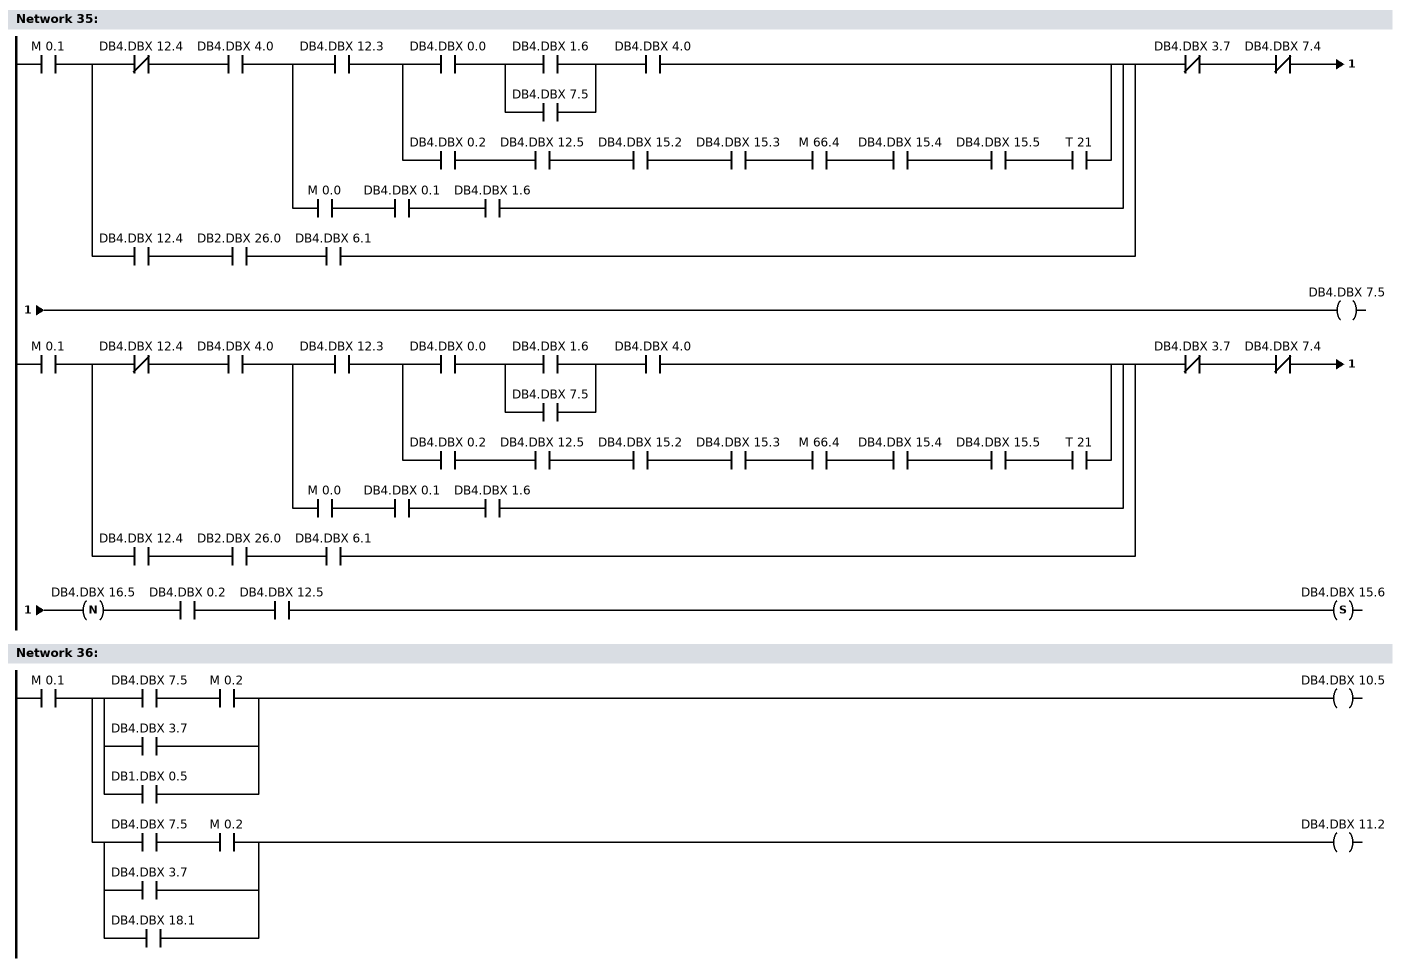
NETWORK
TITLE =
      A     M 0.1;
      A(;
      AN    DB4.DBX 12.4;
      A     DB4.DBX 4.0;
      A(;
      A     DB4.DBX 12.3;
      A(;
      A     DB4.DBX 0.0;
      A(;
      O     DB4.DBX 1.6;
      O     DB4.DBX 7.5;
      );
      A     DB4.DBX 4.0;
      O;
      A     DB4.DBX 0.2;
      A     DB4.DBX 12.5;
      A     DB4.DBX 15.2;
      A     DB4.DBX 15.3;
      A     M 66.4;
      A     DB4.DBX 15.4;
      A     DB4.DBX 15.5;
      A     T 21;
      );
      O;
      A     M 0.0;
      A     DB4.DBX 0.1;
      A     DB4.DBX 1.6;
      );
      O;
      A     DB4.DBX 12.4;
      A     DB2.DBX 26.0;
      A     DB4.DBX 6.1;
      );
      AN    DB4.DBX 3.7;
      AN    DB4.DBX 7.4;
      =     L 0.0;
      A     L 0.0;
      BLD   102;
      =     DB4.DBX 7.5;
      A(;
      A     L 0.0;
      FN    DB4.DBX 16.5;
      );
      A     DB4.DBX 0.2;
      A     DB4.DBX 12.5;
      S     DB4.DBX 15.6;
NETWORK
TITLE =
      A     M 0.1;
      =     L 0.0;
      A     L 0.0;
      A(;
      A     DB4.DBX 7.5;
      A     M 0.2;
      O     DB4.DBX 3.7;
      O     DB1.DBX 0.5;
      );
      =     DB4.DBX 10.5;
      A     L 0.0;
      A(;
      A     DB4.DBX 7.5;
      A     M 0.2;
      O     DB4.DBX 3.7;
      O     DB4.DBX 18.1;
      );
      =     DB4.DBX 11.2;
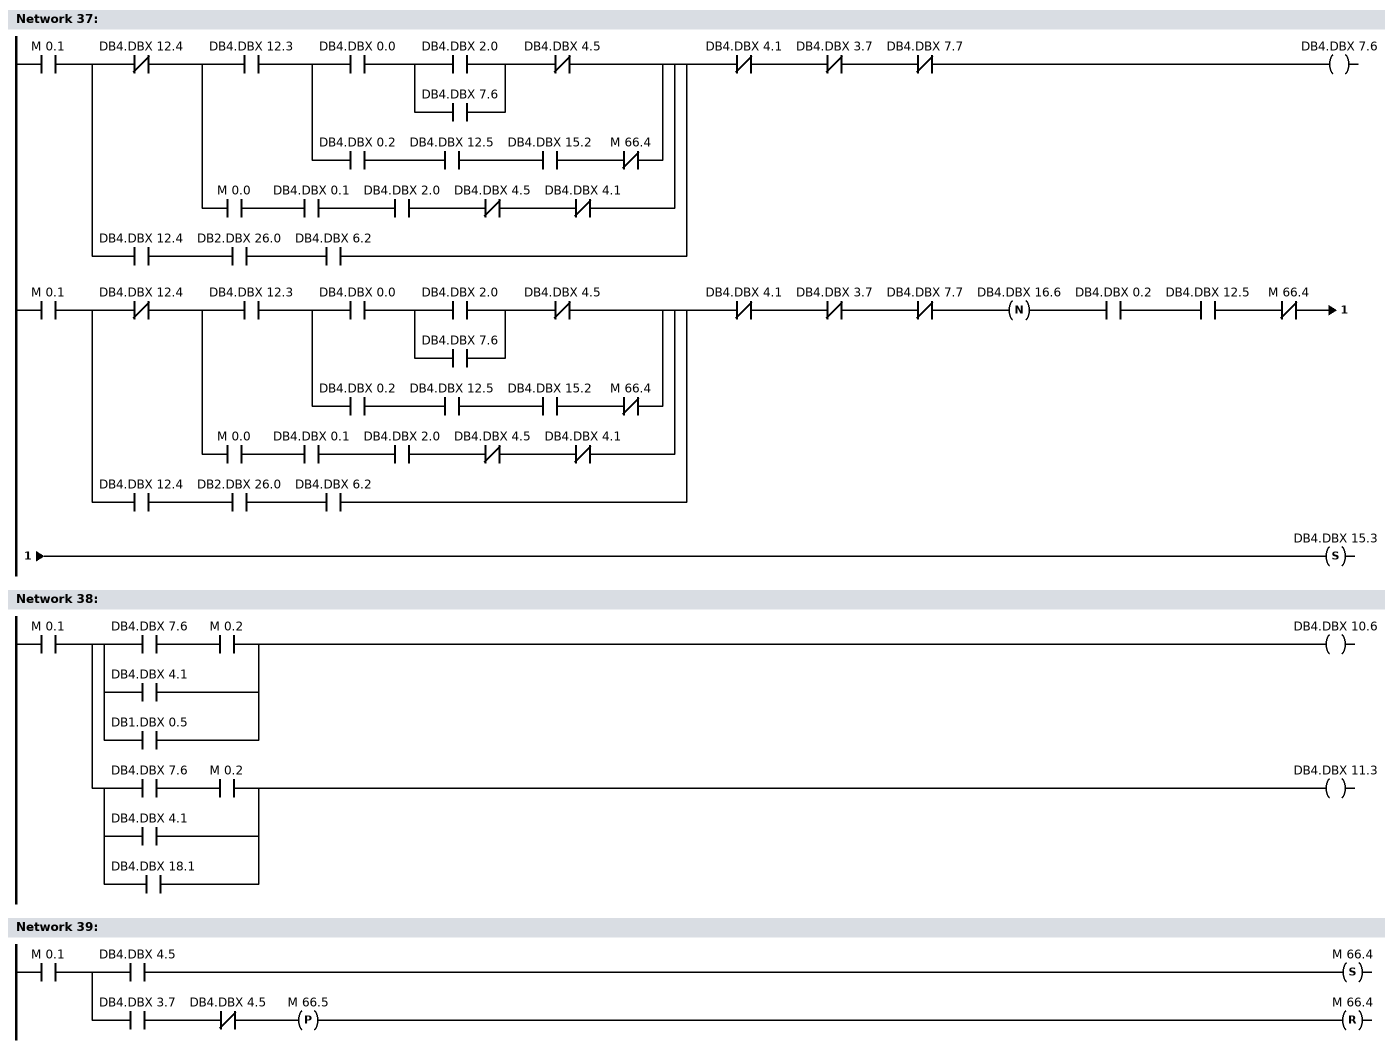
NETWORK
TITLE =
      A     M 0.1;
      A(;
      AN    DB4.DBX 12.4;
      A(;
      A     DB4.DBX 12.3;
      A(;
      A     DB4.DBX 0.0;
      A(;
      O     DB4.DBX 2.0;
      O     DB4.DBX 7.6;
      );
      AN    DB4.DBX 4.5;
      O;
      A     DB4.DBX 0.2;
      A     DB4.DBX 12.5;
      A     DB4.DBX 15.2;
      AN    M 66.4;
      );
      O;
      A     M 0.0;
      A     DB4.DBX 0.1;
      A     DB4.DBX 2.0;
      AN    DB4.DBX 4.5;
      AN    DB4.DBX 4.1;
      );
      O;
      A     DB4.DBX 12.4;
      A     DB2.DBX 26.0;
      A     DB4.DBX 6.2;
      );
      AN    DB4.DBX 4.1;
      AN    DB4.DBX 3.7;
      AN    DB4.DBX 7.7;
      =     L 0.0;
      A     L 0.0;
      BLD   102;
      =     DB4.DBX 7.6;
      A(;
      A     L 0.0;
      FN    DB4.DBX 16.6;
      );
      A     DB4.DBX 0.2;
      A     DB4.DBX 12.5;
      AN    M 66.4;
      S     DB4.DBX 15.3;
NETWORK
TITLE =
      A     M 0.1;
      =     L 0.0;
      A     L 0.0;
      A(;
      A     DB4.DBX 7.6;
      A     M 0.2;
      O     DB4.DBX 4.1;
      O     DB1.DBX 0.5;
      );
      =     DB4.DBX 10.6;
      A     L 0.0;
      A(;
      A     DB4.DBX 7.6;
      A     M 0.2;
      O     DB4.DBX 4.1;
      O     DB4.DBX 18.1;
      );
      =     DB4.DBX 11.3;
NETWORK
TITLE =
      A     M 0.1;
      =     L 0.0;
      A     L 0.0;
      A     DB4.DBX 4.5;
      S     M 66.4;
      A     L 0.0;
      A     DB4.DBX 3.7;
      AN    DB4.DBX 4.5;
      FP    M 66.5;
      R     M 66.4;
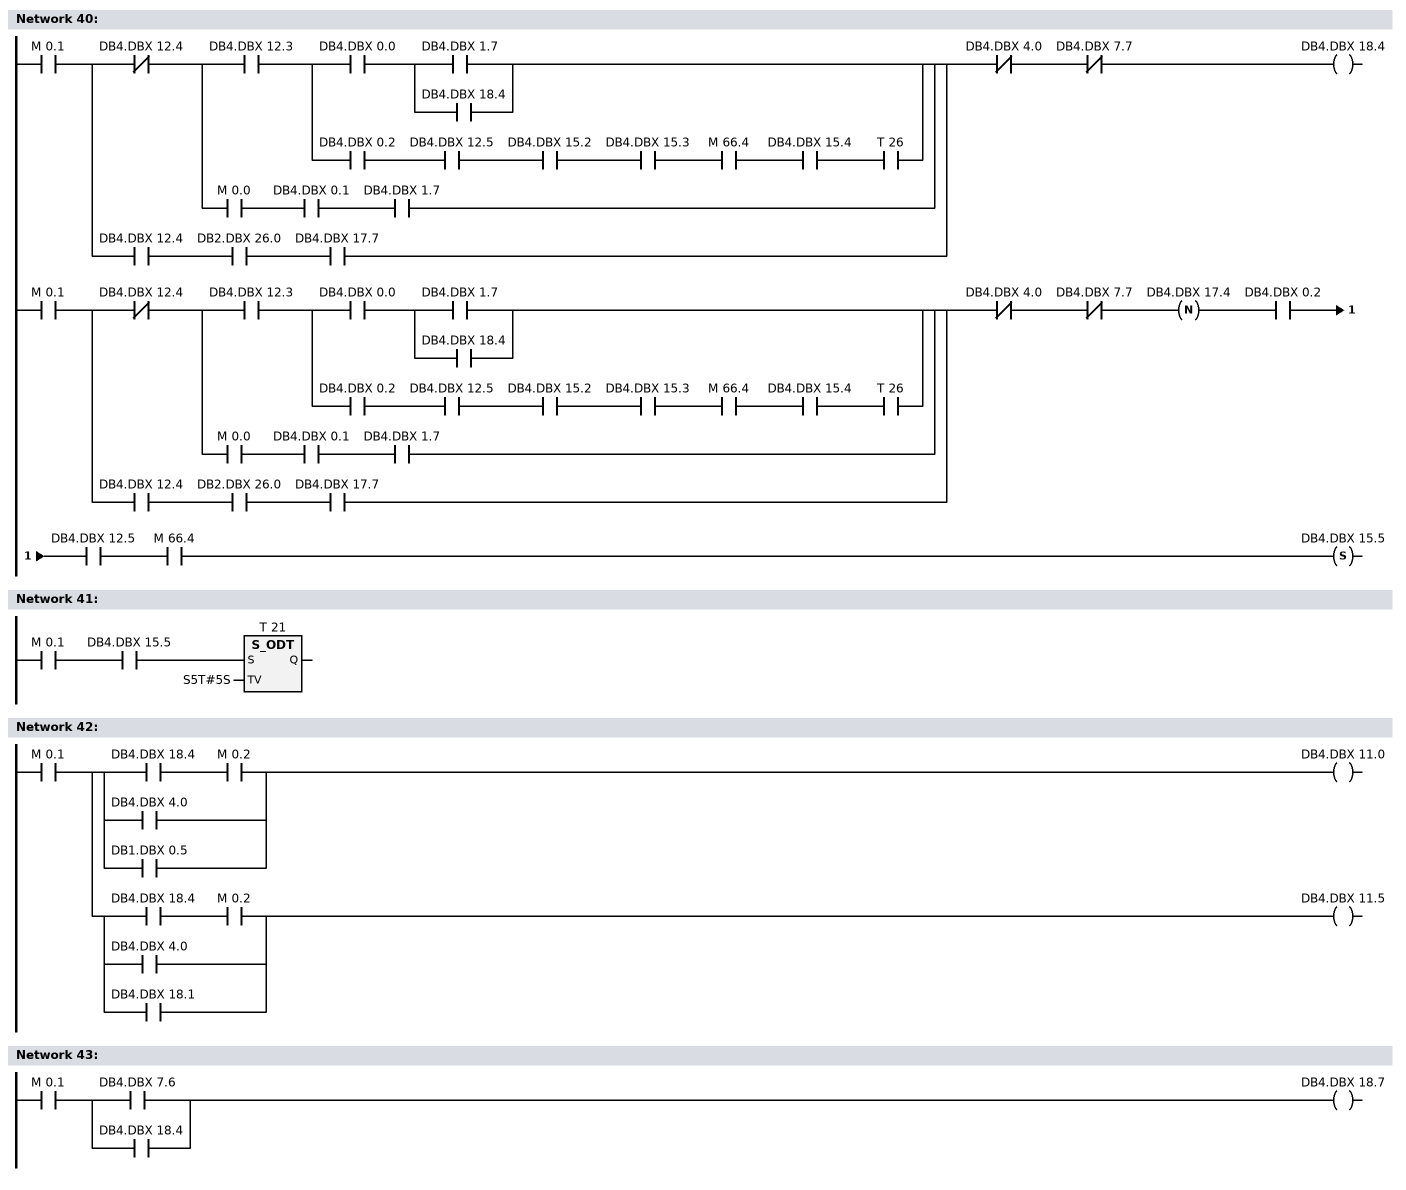
NETWORK
TITLE =
      A     M 0.1;
      A(;
      AN    DB4.DBX 12.4;
      A(;
      A     DB4.DBX 12.3;
      A(;
      A     DB4.DBX 0.0;
      A(;
      O     DB4.DBX 1.7;
      O     DB4.DBX 18.4;
      );
      O;
      A     DB4.DBX 0.2;
      A     DB4.DBX 12.5;
      A     DB4.DBX 15.2;
      A     DB4.DBX 15.3;
      A     M 66.4;
      A     DB4.DBX 15.4;
      A     T 26;
      );
      O;
      A     M 0.0;
      A     DB4.DBX 0.1;
      A     DB4.DBX 1.7;
      );
      O;
      A     DB4.DBX 12.4;
      A     DB2.DBX 26.0;
      A     DB4.DBX 17.7;
      );
      AN    DB4.DBX 4.0;
      AN    DB4.DBX 7.7;
      =     L 0.0;
      A     L 0.0;
      BLD   102;
      =     DB4.DBX 18.4;
      A(;
      A     L 0.0;
      FN    DB4.DBX 17.4;
      );
      A     DB4.DBX 0.2;
      A     DB4.DBX 12.5;
      A     M 66.4;
      S     DB4.DBX 15.5;
NETWORK
TITLE =
      A     M 0.1;
      A     DB4.DBX 15.5;
      L     S5T#5S;
      SD    T 21;
      NOP   0;
      NOP   0;
      NOP   0;
      NOP   0;
NETWORK
TITLE =
      A     M 0.1;
      =     L 0.0;
      A     L 0.0;
      A(;
      A     DB4.DBX 18.4;
      A     M 0.2;
      O     DB4.DBX 4.0;
      O     DB1.DBX 0.5;
      );
      =     DB4.DBX 11.0;
      A     L 0.0;
      A(;
      A     DB4.DBX 18.4;
      A     M 0.2;
      O     DB4.DBX 4.0;
      O     DB4.DBX 18.1;
      );
      =     DB4.DBX 11.5;
NETWORK
TITLE =
      A     M 0.1;
      A(;
      O     DB4.DBX 7.6;
      O     DB4.DBX 18.4;
      );
      =     DB4.DBX 18.7;
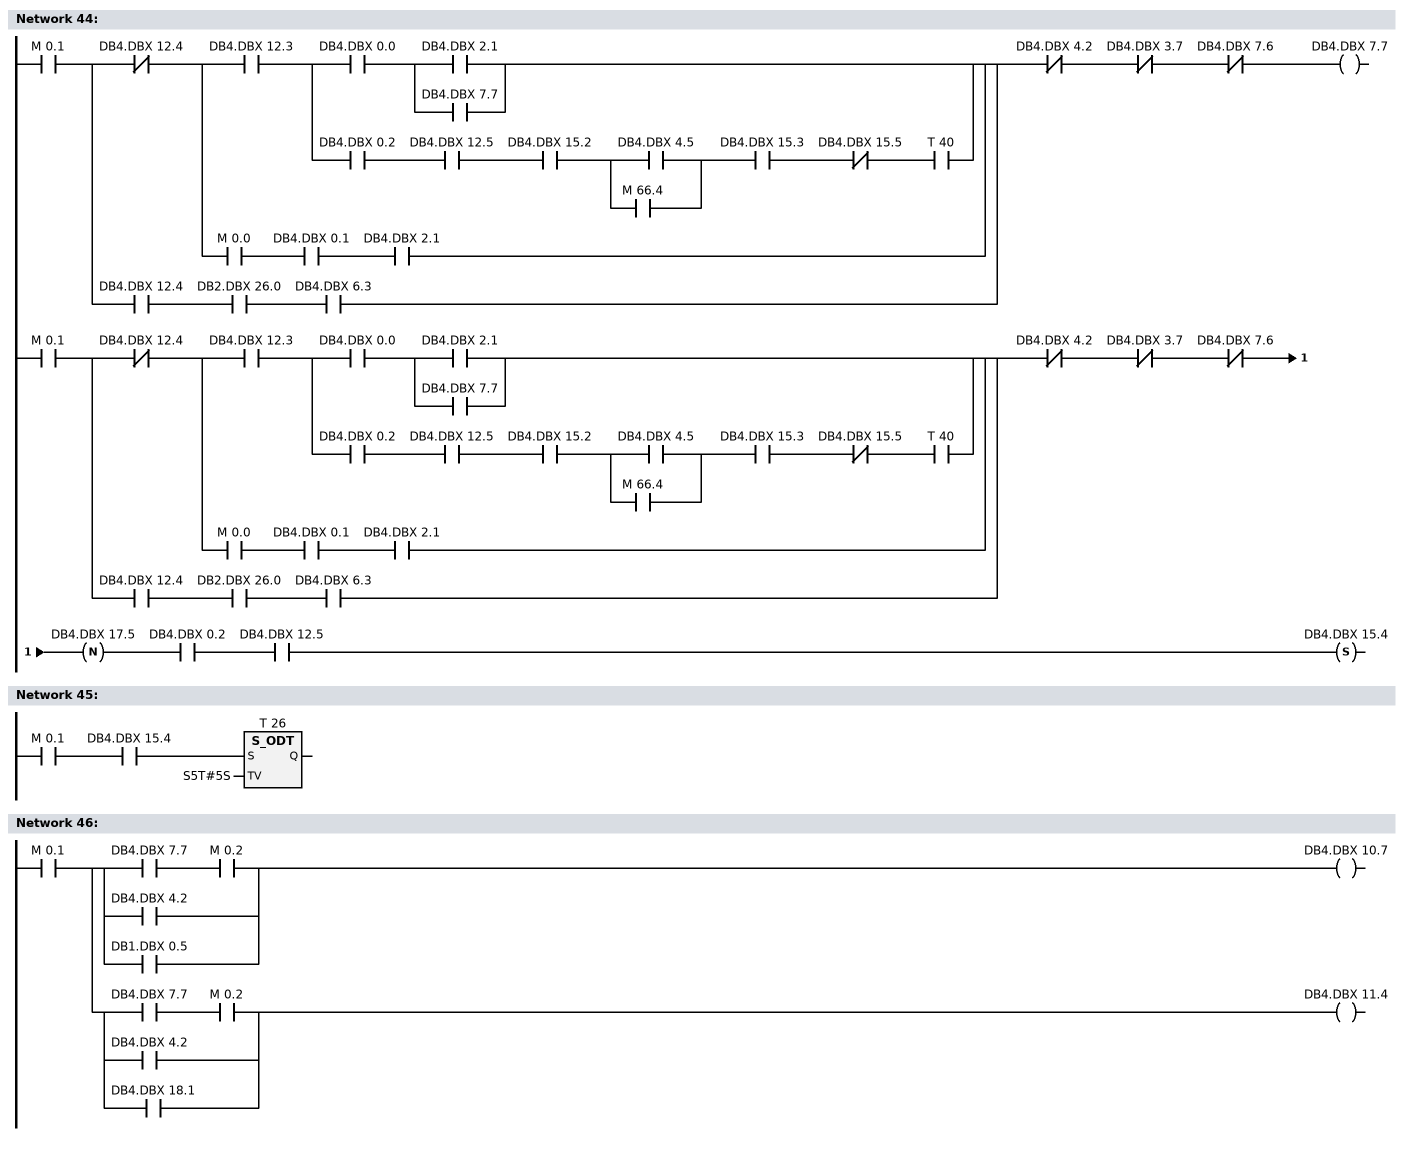
NETWORK
TITLE =
      A     M 0.1;
      A(;
      AN    DB4.DBX 12.4;
      A(;
      A     DB4.DBX 12.3;
      A(;
      A     DB4.DBX 0.0;
      A(;
      O     DB4.DBX 2.1;
      O     DB4.DBX 7.7;
      );
      O;
      A     DB4.DBX 0.2;
      A     DB4.DBX 12.5;
      A     DB4.DBX 15.2;
      A(;
      O     DB4.DBX 4.5;
      O     M 66.4;
      );
      A     DB4.DBX 15.3;
      AN    DB4.DBX 15.5;
      A     T 40;
      );
      O;
      A     M 0.0;
      A     DB4.DBX 0.1;
      A     DB4.DBX 2.1;
      );
      O;
      A     DB4.DBX 12.4;
      A     DB2.DBX 26.0;
      A     DB4.DBX 6.3;
      );
      AN    DB4.DBX 4.2;
      AN    DB4.DBX 3.7;
      AN    DB4.DBX 7.6;
      =     L 0.0;
      A     L 0.0;
      BLD   102;
      =     DB4.DBX 7.7;
      A(;
      A     L 0.0;
      FN    DB4.DBX 17.5;
      );
      A     DB4.DBX 0.2;
      A     DB4.DBX 12.5;
      S     DB4.DBX 15.4;
NETWORK
TITLE =
      A     M 0.1;
      A     DB4.DBX 15.4;
      L     S5T#5S;
      SD    T 26;
      NOP   0;
      NOP   0;
      NOP   0;
      NOP   0;
NETWORK
TITLE =
      A     M 0.1;
      =     L 0.0;
      A     L 0.0;
      A(;
      A     DB4.DBX 7.7;
      A     M 0.2;
      O     DB4.DBX 4.2;
      O     DB1.DBX 0.5;
      );
      =     DB4.DBX 10.7;
      A     L 0.0;
      A(;
      A     DB4.DBX 7.7;
      A     M 0.2;
      O     DB4.DBX 4.2;
      O     DB4.DBX 18.1;
      );
      =     DB4.DBX 11.4;
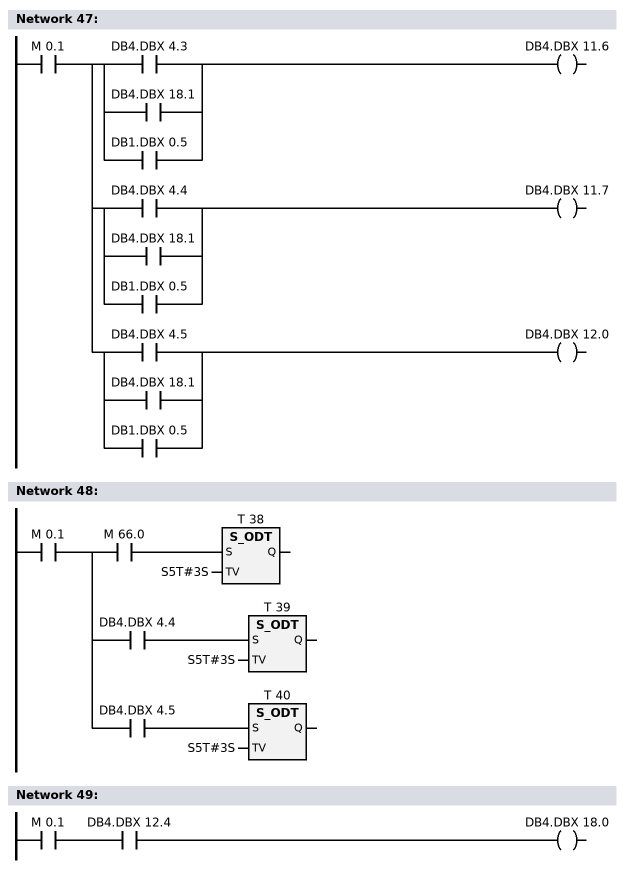
NETWORK
TITLE =
      A     M 0.1;
      =     L 0.0;
      A     L 0.0;
      A(;
      O     DB4.DBX 4.3;
      O     DB4.DBX 18.1;
      O     DB1.DBX 0.5;
      );
      =     DB4.DBX 11.6;
      A     L 0.0;
      A(;
      O     DB4.DBX 4.4;
      O     DB4.DBX 18.1;
      O     DB1.DBX 0.5;
      );
      =     DB4.DBX 11.7;
      A     L 0.0;
      A(;
      O     DB4.DBX 4.5;
      O     DB4.DBX 18.1;
      O     DB1.DBX 0.5;
      );
      =     DB4.DBX 12.0;
NETWORK
TITLE =
      A     M 0.1;
      =     L 0.0;
      A     L 0.0;
      A     M 66.0;
      L     S5T#3S;
      SD    T 38;
      NOP   0;
      NOP   0;
      NOP   0;
      NOP   0;
      A     L 0.0;
      A     DB4.DBX 4.4;
      L     S5T#3S;
      SD    T 39;
      NOP   0;
      NOP   0;
      NOP   0;
      NOP   0;
      A     L 0.0;
      A     DB4.DBX 4.5;
      L     S5T#3S;
      SD    T 40;
      NOP   0;
      NOP   0;
      NOP   0;
      NOP   0;
NETWORK
TITLE =
      A     M 0.1;
      A     DB4.DBX 12.4;
      =     DB4.DBX 18.0;
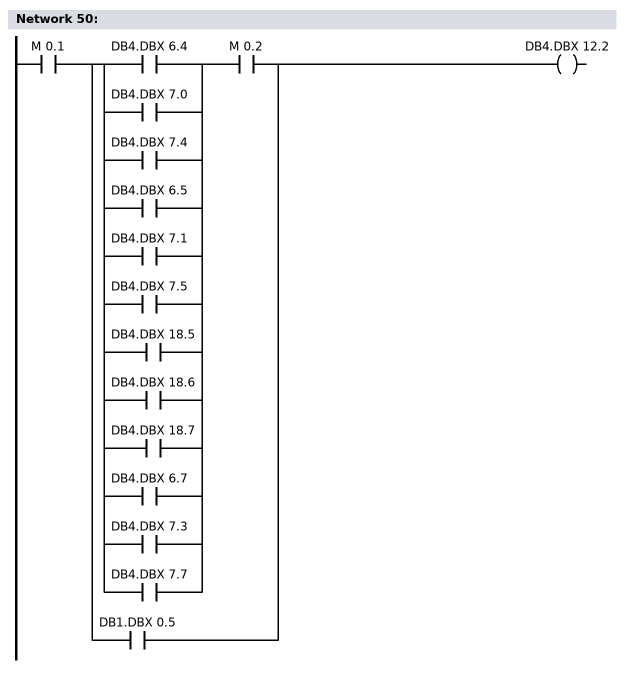
NETWORK
TITLE =
      A     M 0.1;
      A(;
      A(;
      O     DB4.DBX 6.4;
      O     DB4.DBX 7.0;
      O     DB4.DBX 7.4;
      O     DB4.DBX 6.5;
      O     DB4.DBX 7.1;
      O     DB4.DBX 7.5;
      O     DB4.DBX 18.5;
      O     DB4.DBX 18.6;
      O     DB4.DBX 18.7;
      O     DB4.DBX 6.7;
      O     DB4.DBX 7.3;
      O     DB4.DBX 7.7;
      );
      A     M 0.2;
      O     DB1.DBX 0.5;
      );
      =     DB4.DBX 12.2;
END_FUNCTION

FUNCTION FC 10 : VOID
AUTHOR : Arun_Ram
VERSION : 0.1
BEGIN
// (block stored without names or comments; labels and parameter names are numbered)
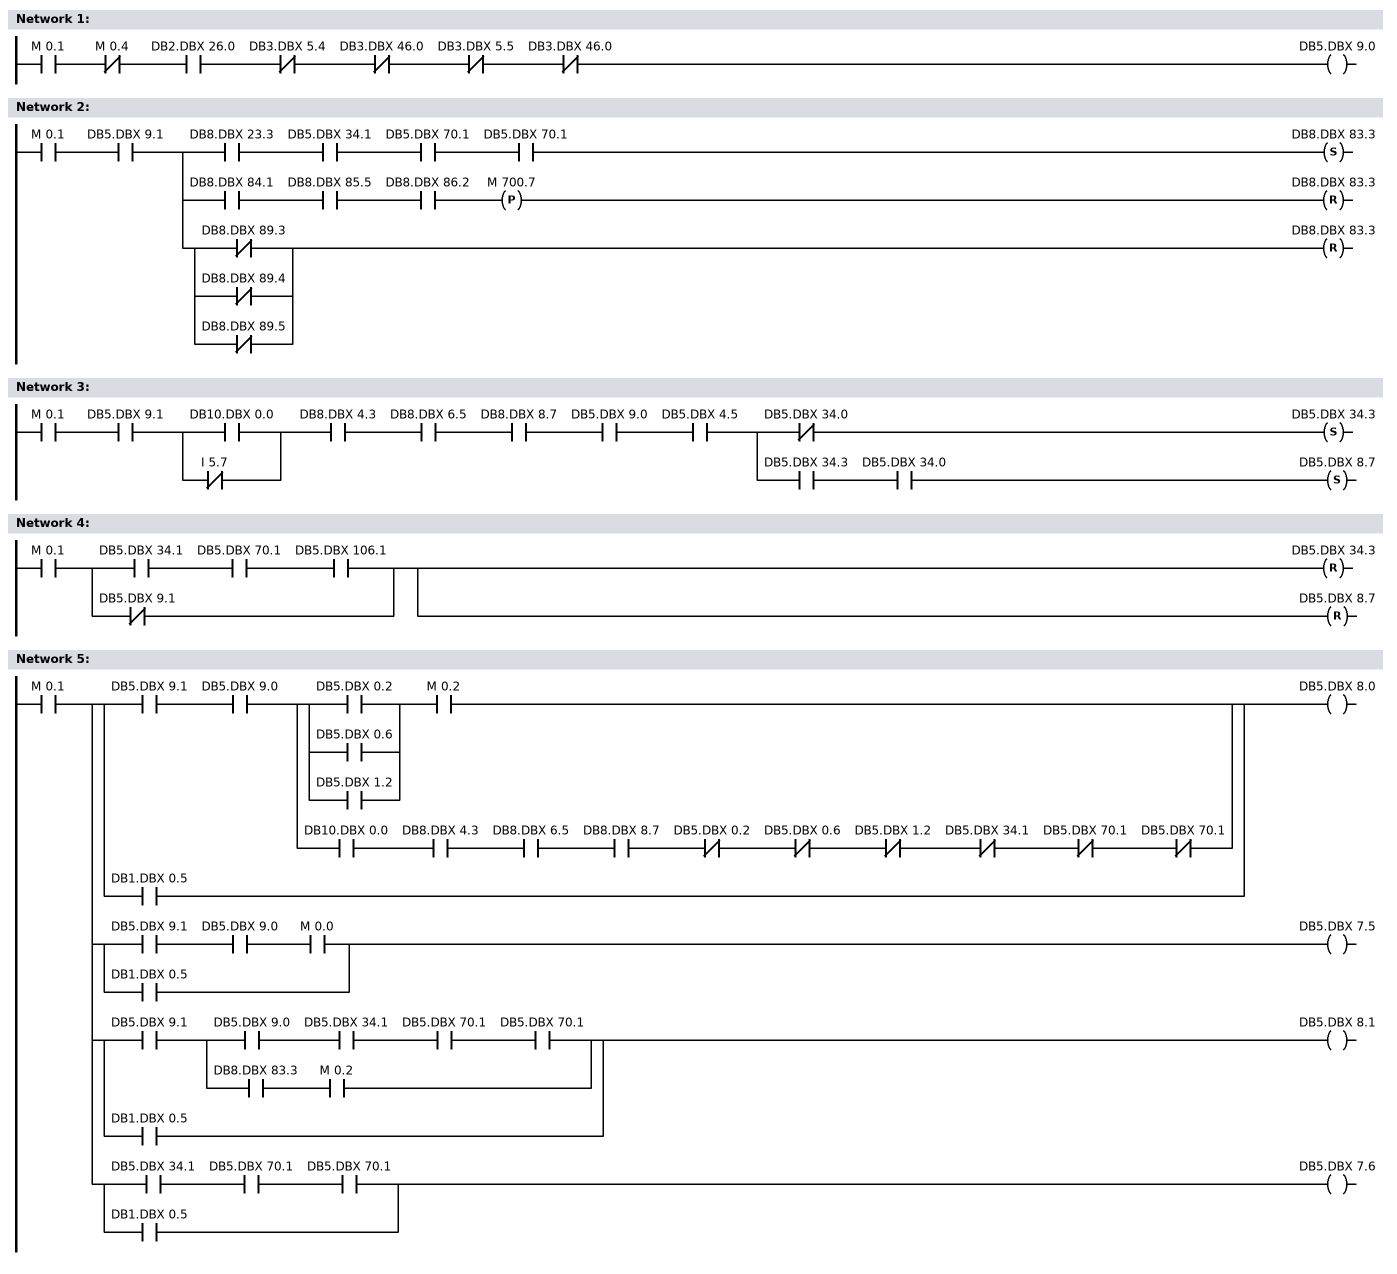
NETWORK
TITLE =
      A     M 0.1;
      AN    M 0.4;
      A     DB2.DBX 26.0;
      AN    DB3.DBX 5.4;
      AN    DB3.DBX 46.0;
      AN    DB3.DBX 5.5;
      AN    DB3.DBX 46.0;
      =     DB5.DBX 9.0;
NETWORK
TITLE =
      A     M 0.1;
      A     DB5.DBX 9.1;
      =     L 0.0;
      A     L 0.0;
      A     DB8.DBX 23.3;
      A     DB5.DBX 34.1;
      A     DB5.DBX 70.1;
      A     DB5.DBX 70.1;
      S     DB8.DBX 83.3;
      A     L 0.0;
      A     DB8.DBX 84.1;
      A     DB8.DBX 85.5;
      A     DB8.DBX 86.2;
      FP    M 700.7;
      R     DB8.DBX 83.3;
      A     L 0.0;
      A(;
      ON    DB8.DBX 89.3;
      ON    DB8.DBX 89.4;
      ON    DB8.DBX 89.5;
      );
      R     DB8.DBX 83.3;
NETWORK
TITLE =
      A     M 0.1;
      A     DB5.DBX 9.1;
      A(;
      O     DB10.DBX 0.0;
      ON    I 5.7;
      );
      A     DB8.DBX 4.3;
      A     DB8.DBX 6.5;
      A     DB8.DBX 8.7;
      A     DB5.DBX 9.0;
      A     DB5.DBX 4.5;
      =     L 0.0;
      A     L 0.0;
      AN    DB5.DBX 34.0;
      S     DB5.DBX 34.3;
      A     L 0.0;
      A     DB5.DBX 34.3;
      A     DB5.DBX 34.0;
      S     DB5.DBX 8.7;
NETWORK
TITLE =
      A     M 0.1;
      A(;
      A     DB5.DBX 34.1;
      A     DB5.DBX 70.1;
      A     DB5.DBX 106.1;
      ON    DB5.DBX 9.1;
      );
      R     DB5.DBX 34.3;
      R     DB5.DBX 8.7;
NETWORK
TITLE =
      A     M 0.1;
      =     L 0.0;
      A     L 0.0;
      A(;
      A     DB5.DBX 9.1;
      A     DB5.DBX 9.0;
      A(;
      A(;
      O     DB5.DBX 0.2;
      O     DB5.DBX 0.6;
      O     DB5.DBX 1.2;
      );
      A     M 0.2;
      O;
      A     DB10.DBX 0.0;
      A     DB8.DBX 4.3;
      A     DB8.DBX 6.5;
      A     DB8.DBX 8.7;
      AN    DB5.DBX 0.2;
      AN    DB5.DBX 0.6;
      AN    DB5.DBX 1.2;
      AN    DB5.DBX 34.1;
      AN    DB5.DBX 70.1;
      AN    DB5.DBX 70.1;
      );
      O     DB1.DBX 0.5;
      );
      =     DB5.DBX 8.0;
      A     L 0.0;
      A(;
      A     DB5.DBX 9.1;
      A     DB5.DBX 9.0;
      A     M 0.0;
      O     DB1.DBX 0.5;
      );
      =     DB5.DBX 7.5;
      A     L 0.0;
      A(;
      A     DB5.DBX 9.1;
      A(;
      A     DB5.DBX 9.0;
      A     DB5.DBX 34.1;
      A     DB5.DBX 70.1;
      A     DB5.DBX 70.1;
      O;
      A     DB8.DBX 83.3;
      A     M 0.2;
      );
      O     DB1.DBX 0.5;
      );
      =     DB5.DBX 8.1;
      A     L 0.0;
      A(;
      A     DB5.DBX 34.1;
      A     DB5.DBX 70.1;
      A     DB5.DBX 70.1;
      O     DB1.DBX 0.5;
      );
      =     DB5.DBX 7.6;
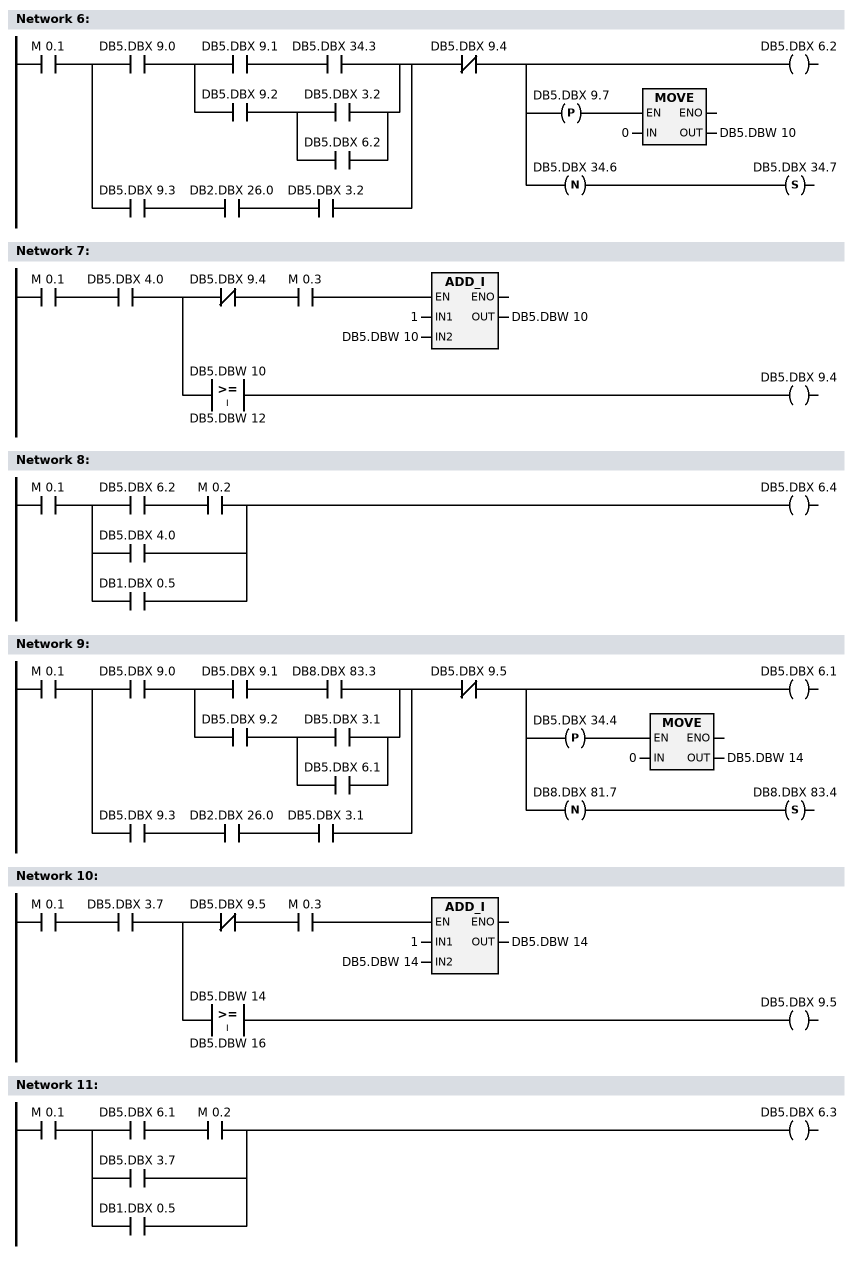
NETWORK
TITLE =
      A     M 0.1;
      A(;
      A     DB5.DBX 9.0;
      A(;
      A     DB5.DBX 9.1;
      A     DB5.DBX 34.3;
      O;
      A     DB5.DBX 9.2;
      A(;
      O     DB5.DBX 3.2;
      O     DB5.DBX 6.2;
      );
      );
      O;
      A     DB5.DBX 9.3;
      A     DB2.DBX 26.0;
      A     DB5.DBX 3.2;
      );
      AN    DB5.DBX 9.4;
      =     L 0.0;
      A     L 0.0;
      BLD   102;
      =     DB5.DBX 6.2;
      A     L 0.0;
      FP    DB5.DBX 9.7;
      JNB   M001;
      L     0;
      T     DB5.DBW 10;
M001: NOP   0;
      A     L 0.0;
      FN    DB5.DBX 34.6;
      S     DB5.DBX 34.7;
NETWORK
TITLE =
      A     M 0.1;
      A     DB5.DBX 4.0;
      =     L 0.0;
      A     L 0.0;
      AN    DB5.DBX 9.4;
      A     M 0.3;
      JNB   M002;
      L     1;
      L     DB5.DBW 10;
      +I;
      T     DB5.DBW 10;
M002: NOP   0;
      A     L 0.0;
      A(;
      L     DB5.DBW 10;
      L     DB5.DBW 12;
      >=I;
      );
      =     DB5.DBX 9.4;
NETWORK
TITLE =
      A     M 0.1;
      A(;
      A     DB5.DBX 6.2;
      A     M 0.2;
      O     DB5.DBX 4.0;
      O     DB1.DBX 0.5;
      );
      =     DB5.DBX 6.4;
NETWORK
TITLE =
      A     M 0.1;
      A(;
      A     DB5.DBX 9.0;
      A(;
      A     DB5.DBX 9.1;
      A     DB8.DBX 83.3;
      O;
      A     DB5.DBX 9.2;
      A(;
      O     DB5.DBX 3.1;
      O     DB5.DBX 6.1;
      );
      );
      O;
      A     DB5.DBX 9.3;
      A     DB2.DBX 26.0;
      A     DB5.DBX 3.1;
      );
      AN    DB5.DBX 9.5;
      =     L 0.0;
      A     L 0.0;
      BLD   102;
      =     DB5.DBX 6.1;
      A     L 0.0;
      FP    DB5.DBX 34.4;
      JNB   M003;
      L     0;
      T     DB5.DBW 14;
M003: NOP   0;
      A     L 0.0;
      FN    DB8.DBX 81.7;
      S     DB8.DBX 83.4;
NETWORK
TITLE =
      A     M 0.1;
      A     DB5.DBX 3.7;
      =     L 0.0;
      A     L 0.0;
      AN    DB5.DBX 9.5;
      A     M 0.3;
      JNB   M004;
      L     1;
      L     DB5.DBW 14;
      +I;
      T     DB5.DBW 14;
M004: NOP   0;
      A     L 0.0;
      A(;
      L     DB5.DBW 14;
      L     DB5.DBW 16;
      >=I;
      );
      =     DB5.DBX 9.5;
NETWORK
TITLE =
      A     M 0.1;
      A(;
      A     DB5.DBX 6.1;
      A     M 0.2;
      O     DB5.DBX 3.7;
      O     DB1.DBX 0.5;
      );
      =     DB5.DBX 6.3;
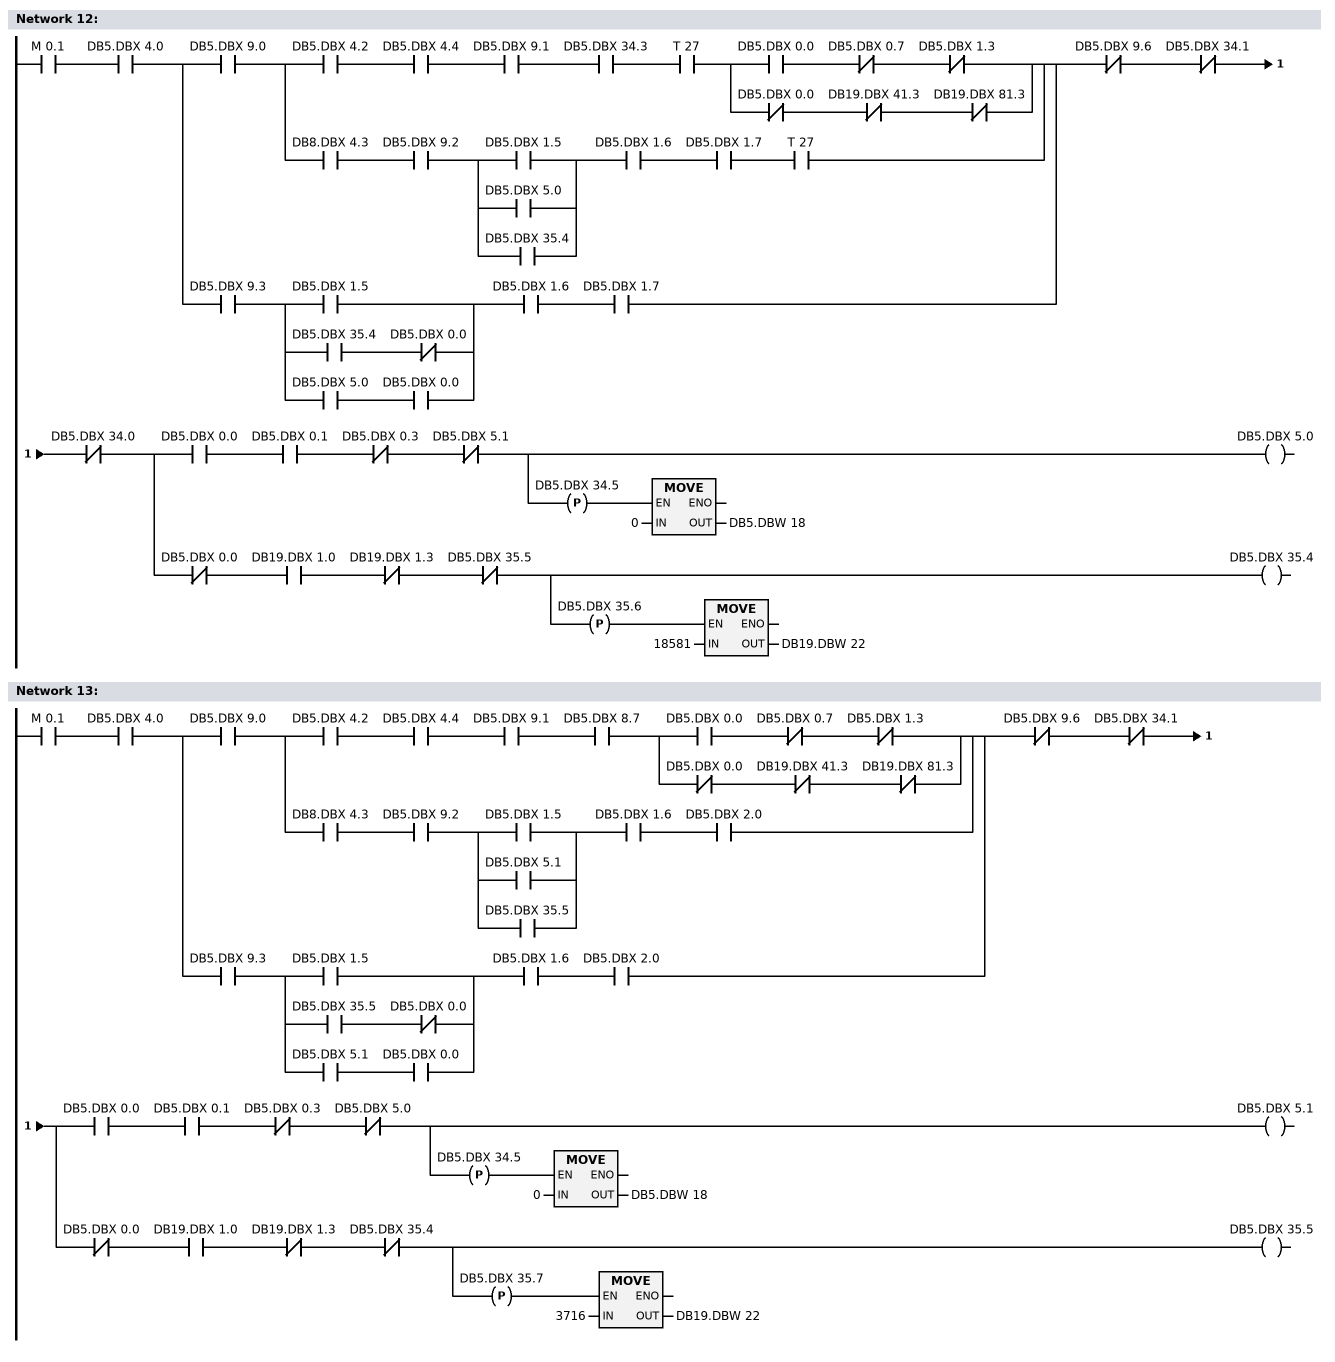
NETWORK
TITLE =
      A     M 0.1;
      A     DB5.DBX 4.0;
      A(;
      A     DB5.DBX 9.0;
      A(;
      A     DB5.DBX 4.2;
      A     DB5.DBX 4.4;
      A     DB5.DBX 9.1;
      A     DB5.DBX 34.3;
      A     T 27;
      A(;
      A     DB5.DBX 0.0;
      AN    DB5.DBX 0.7;
      AN    DB5.DBX 1.3;
      O;
      AN    DB5.DBX 0.0;
      AN    DB19.DBX 41.3;
      AN    DB19.DBX 81.3;
      );
      O;
      A     DB8.DBX 4.3;
      A     DB5.DBX 9.2;
      A(;
      O     DB5.DBX 1.5;
      O     DB5.DBX 5.0;
      O     DB5.DBX 35.4;
      );
      A     DB5.DBX 1.6;
      A     DB5.DBX 1.7;
      A     T 27;
      );
      O;
      A     DB5.DBX 9.3;
      A(;
      O     DB5.DBX 1.5;
      O;
      A     DB5.DBX 35.4;
      AN    DB5.DBX 0.0;
      O;
      A     DB5.DBX 5.0;
      A     DB5.DBX 0.0;
      );
      A     DB5.DBX 1.6;
      A     DB5.DBX 1.7;
      );
      AN    DB5.DBX 9.6;
      AN    DB5.DBX 34.1;
      AN    DB5.DBX 34.0;
      =     L 0.0;
      A     L 0.0;
      A     DB5.DBX 0.0;
      A     DB5.DBX 0.1;
      AN    DB5.DBX 0.3;
      AN    DB5.DBX 5.1;
      =     L 0.1;
      A     L 0.1;
      BLD   102;
      =     DB5.DBX 5.0;
      A     L 0.1;
      FP    DB5.DBX 34.5;
      JNB   M005;
      L     0;
      T     DB5.DBW 18;
M005: NOP   0;
      A     L 0.0;
      AN    DB5.DBX 0.0;
      A     DB19.DBX 1.0;
      AN    DB19.DBX 1.3;
      AN    DB5.DBX 35.5;
      =     L 0.1;
      A     L 0.1;
      BLD   102;
      =     DB5.DBX 35.4;
      A     L 0.1;
      FP    DB5.DBX 35.6;
      JNB   M006;
      L     18581;
      T     DB19.DBW 22;
M006: NOP   0;
NETWORK
TITLE =
      A     M 0.1;
      A     DB5.DBX 4.0;
      A(;
      A     DB5.DBX 9.0;
      A(;
      A     DB5.DBX 4.2;
      A     DB5.DBX 4.4;
      A     DB5.DBX 9.1;
      A     DB5.DBX 8.7;
      A(;
      A     DB5.DBX 0.0;
      AN    DB5.DBX 0.7;
      AN    DB5.DBX 1.3;
      O;
      AN    DB5.DBX 0.0;
      AN    DB19.DBX 41.3;
      AN    DB19.DBX 81.3;
      );
      O;
      A     DB8.DBX 4.3;
      A     DB5.DBX 9.2;
      A(;
      O     DB5.DBX 1.5;
      O     DB5.DBX 5.1;
      O     DB5.DBX 35.5;
      );
      A     DB5.DBX 1.6;
      A     DB5.DBX 2.0;
      );
      O;
      A     DB5.DBX 9.3;
      A(;
      O     DB5.DBX 1.5;
      O;
      A     DB5.DBX 35.5;
      AN    DB5.DBX 0.0;
      O;
      A     DB5.DBX 5.1;
      A     DB5.DBX 0.0;
      );
      A     DB5.DBX 1.6;
      A     DB5.DBX 2.0;
      );
      AN    DB5.DBX 9.6;
      AN    DB5.DBX 34.1;
      =     L 0.0;
      A     L 0.0;
      A     DB5.DBX 0.0;
      A     DB5.DBX 0.1;
      AN    DB5.DBX 0.3;
      AN    DB5.DBX 5.0;
      =     L 0.1;
      A     L 0.1;
      BLD   102;
      =     DB5.DBX 5.1;
      A     L 0.1;
      FP    DB5.DBX 34.5;
      JNB   M007;
      L     0;
      T     DB5.DBW 18;
M007: NOP   0;
      A     L 0.0;
      AN    DB5.DBX 0.0;
      A     DB19.DBX 1.0;
      AN    DB19.DBX 1.3;
      AN    DB5.DBX 35.4;
      =     L 0.1;
      A     L 0.1;
      BLD   102;
      =     DB5.DBX 35.5;
      A     L 0.1;
      FP    DB5.DBX 35.7;
      JNB   M008;
      L     3716;
      T     DB19.DBW 22;
M008: NOP   0;
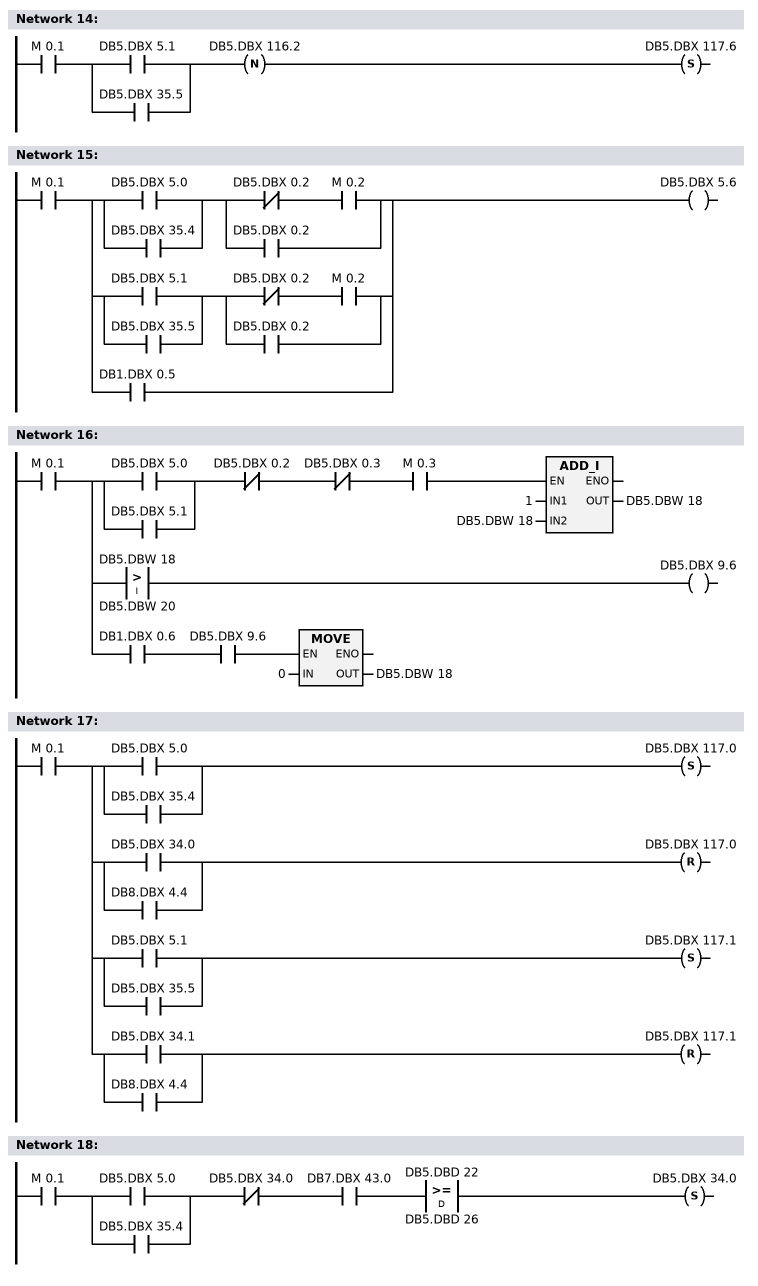
NETWORK
TITLE =
      A     M 0.1;
      A(;
      O     DB5.DBX 5.1;
      O     DB5.DBX 35.5;
      );
      FN    DB5.DBX 116.2;
      S     DB5.DBX 117.6;
NETWORK
TITLE =
      A     M 0.1;
      A(;
      A(;
      O     DB5.DBX 5.0;
      O     DB5.DBX 35.4;
      );
      A(;
      AN    DB5.DBX 0.2;
      A     M 0.2;
      O     DB5.DBX 0.2;
      );
      O;
      A(;
      O     DB5.DBX 5.1;
      O     DB5.DBX 35.5;
      );
      A(;
      AN    DB5.DBX 0.2;
      A     M 0.2;
      O     DB5.DBX 0.2;
      );
      O     DB1.DBX 0.5;
      );
      =     DB5.DBX 5.6;
NETWORK
TITLE =
      A     M 0.1;
      =     L 0.0;
      A     L 0.0;
      A(;
      O     DB5.DBX 5.0;
      O     DB5.DBX 5.1;
      );
      AN    DB5.DBX 0.2;
      AN    DB5.DBX 0.3;
      A     M 0.3;
      JNB   M009;
      L     1;
      L     DB5.DBW 18;
      +I;
      T     DB5.DBW 18;
M009: NOP   0;
      A     L 0.0;
      A(;
      L     DB5.DBW 18;
      L     DB5.DBW 20;
      >I;
      );
      =     DB5.DBX 9.6;
      A     L 0.0;
      A     DB1.DBX 0.6;
      A     DB5.DBX 9.6;
      JNB   M010;
      L     0;
      T     DB5.DBW 18;
M010: NOP   0;
NETWORK
TITLE =
      A     M 0.1;
      =     L 0.0;
      A     L 0.0;
      A(;
      O     DB5.DBX 5.0;
      O     DB5.DBX 35.4;
      );
      S     DB5.DBX 117.0;
      A     L 0.0;
      A(;
      O     DB5.DBX 34.0;
      O     DB8.DBX 4.4;
      );
      R     DB5.DBX 117.0;
      A     L 0.0;
      A(;
      O     DB5.DBX 5.1;
      O     DB5.DBX 35.5;
      );
      S     DB5.DBX 117.1;
      A     L 0.0;
      A(;
      O     DB5.DBX 34.1;
      O     DB8.DBX 4.4;
      );
      R     DB5.DBX 117.1;
NETWORK
TITLE =
      A     M 0.1;
      A(;
      O     DB5.DBX 5.0;
      O     DB5.DBX 35.4;
      );
      AN    DB5.DBX 34.0;
      A     DB7.DBX 43.0;
      A(;
      L     DB5.DBD 22;
      L     DB5.DBD 26;
      >=D;
      );
      S     DB5.DBX 34.0;
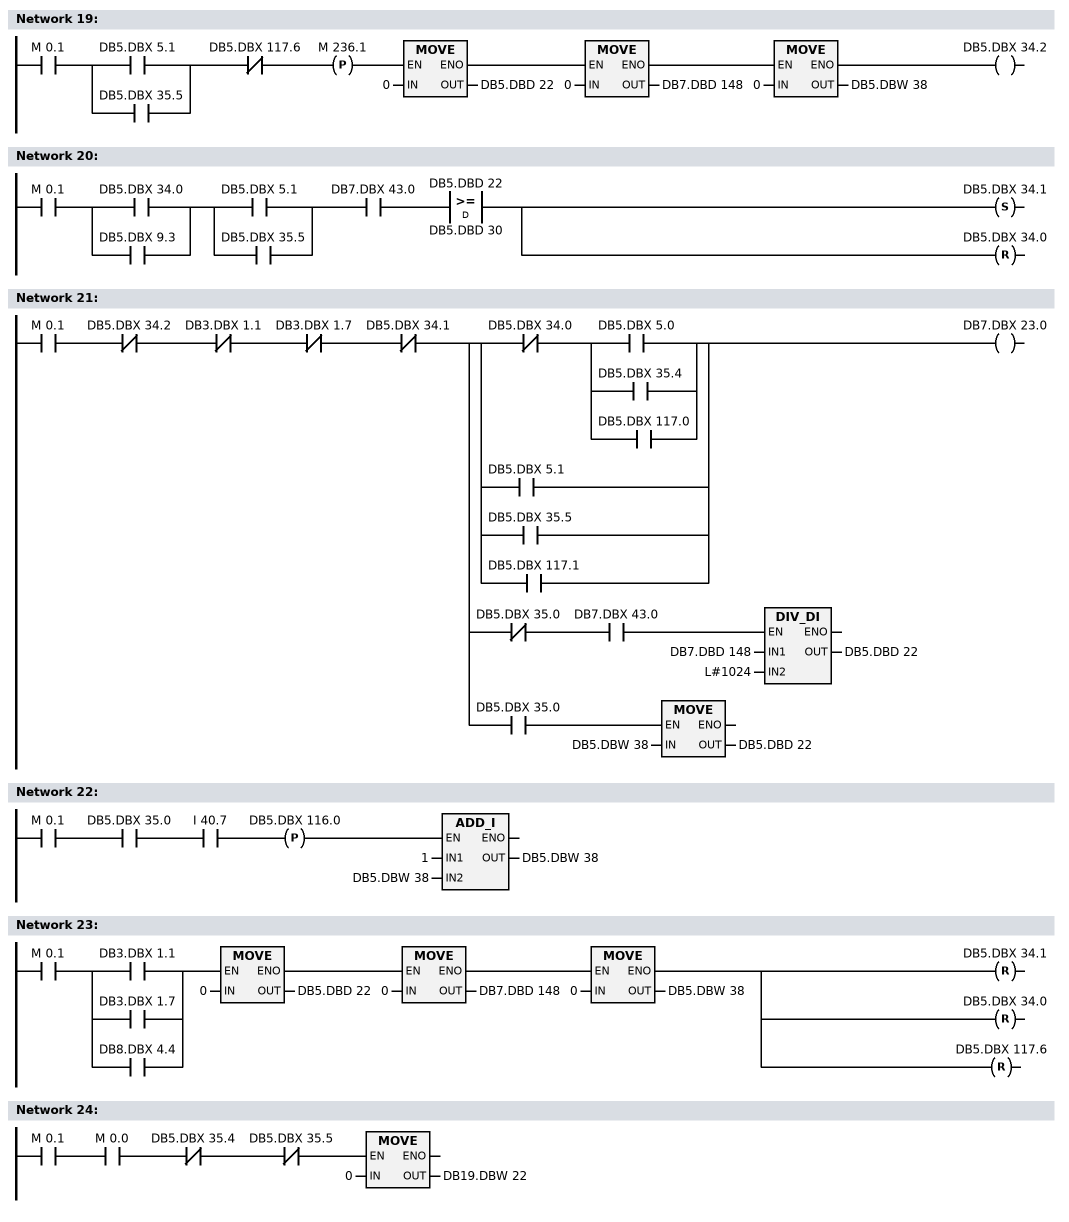
NETWORK
TITLE =
      A(;
      A(;
      A     M 0.1;
      A(;
      O     DB5.DBX 5.1;
      O     DB5.DBX 35.5;
      );
      AN    DB5.DBX 117.6;
      FP    M 236.1;
      JNB   M011;
      L     0;
      T     DB5.DBD 22;
      SET;
      SAVE;
      CLR;
M011: A     BR;
      );
      JNB   M012;
      L     0;
      T     DB7.DBD 148;
      SET;
      SAVE;
      CLR;
M012: A     BR;
      );
      JNB   M013;
      L     0;
      T     DB5.DBW 38;
      SET;
      SAVE;
      CLR;
M013: A     BR;
      =     DB5.DBX 34.2;
NETWORK
TITLE =
      A     M 0.1;
      A(;
      O     DB5.DBX 34.0;
      O     DB5.DBX 9.3;
      );
      A(;
      O     DB5.DBX 5.1;
      O     DB5.DBX 35.5;
      );
      A     DB7.DBX 43.0;
      A(;
      L     DB5.DBD 22;
      L     DB5.DBD 30;
      >=D;
      );
      S     DB5.DBX 34.1;
      R     DB5.DBX 34.0;
NETWORK
TITLE =
      A     M 0.1;
      AN    DB5.DBX 34.2;
      AN    DB3.DBX 1.1;
      AN    DB3.DBX 1.7;
      AN    DB5.DBX 34.1;
      =     L 0.0;
      A     L 0.0;
      A(;
      AN    DB5.DBX 34.0;
      A(;
      O     DB5.DBX 5.0;
      O     DB5.DBX 35.4;
      O     DB5.DBX 117.0;
      );
      O     DB5.DBX 5.1;
      O     DB5.DBX 35.5;
      O     DB5.DBX 117.1;
      );
      =     DB7.DBX 23.0;
      A     L 0.0;
      AN    DB5.DBX 35.0;
      A     DB7.DBX 43.0;
      JNB   M014;
      L     DB7.DBD 148;
      L     L#1024;
      /D;
      T     DB5.DBD 22;
M014: NOP   0;
      A     L 0.0;
      A     DB5.DBX 35.0;
      JNB   M015;
      L     DB5.DBW 38;
      T     DB5.DBD 22;
M015: NOP   0;
NETWORK
TITLE =
      A     M 0.1;
      A     DB5.DBX 35.0;
      A     I 40.7;
      FP    DB5.DBX 116.0;
      JNB   M016;
      L     1;
      L     DB5.DBW 38;
      +I;
      T     DB5.DBW 38;
M016: NOP   0;
NETWORK
TITLE =
      A(;
      A(;
      A     M 0.1;
      A(;
      O     DB3.DBX 1.1;
      O     DB3.DBX 1.7;
      O     DB8.DBX 4.4;
      );
      JNB   M017;
      L     0;
      T     DB5.DBD 22;
      SET;
      SAVE;
      CLR;
M017: A     BR;
      );
      JNB   M018;
      L     0;
      T     DB7.DBD 148;
      SET;
      SAVE;
      CLR;
M018: A     BR;
      );
      JNB   M019;
      L     0;
      T     DB5.DBW 38;
      SET;
      SAVE;
      CLR;
M019: A     BR;
      R     DB5.DBX 34.1;
      R     DB5.DBX 34.0;
      R     DB5.DBX 117.6;
NETWORK
TITLE =
      A     M 0.1;
      A     M 0.0;
      AN    DB5.DBX 35.4;
      AN    DB5.DBX 35.5;
      JNB   M020;
      L     0;
      T     DB19.DBW 22;
M020: NOP   0;
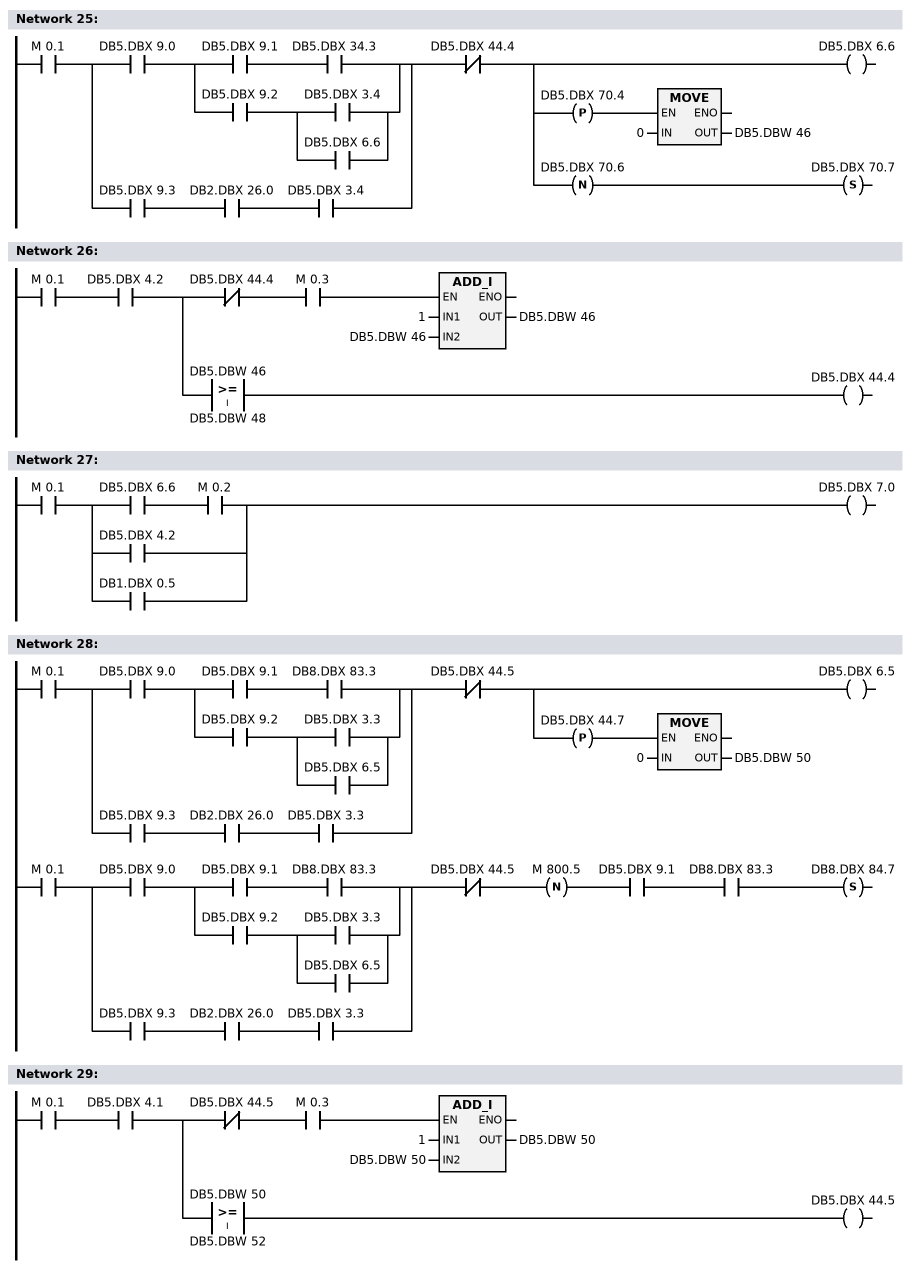
NETWORK
TITLE =
      A     M 0.1;
      A(;
      A     DB5.DBX 9.0;
      A(;
      A     DB5.DBX 9.1;
      A     DB5.DBX 34.3;
      O;
      A     DB5.DBX 9.2;
      A(;
      O     DB5.DBX 3.4;
      O     DB5.DBX 6.6;
      );
      );
      O;
      A     DB5.DBX 9.3;
      A     DB2.DBX 26.0;
      A     DB5.DBX 3.4;
      );
      AN    DB5.DBX 44.4;
      =     L 0.0;
      A     L 0.0;
      BLD   102;
      =     DB5.DBX 6.6;
      A     L 0.0;
      FP    DB5.DBX 70.4;
      JNB   M021;
      L     0;
      T     DB5.DBW 46;
M021: NOP   0;
      A     L 0.0;
      FN    DB5.DBX 70.6;
      S     DB5.DBX 70.7;
NETWORK
TITLE =
      A     M 0.1;
      A     DB5.DBX 4.2;
      =     L 0.0;
      A     L 0.0;
      AN    DB5.DBX 44.4;
      A     M 0.3;
      JNB   M022;
      L     1;
      L     DB5.DBW 46;
      +I;
      T     DB5.DBW 46;
M022: NOP   0;
      A     L 0.0;
      A(;
      L     DB5.DBW 46;
      L     DB5.DBW 48;
      >=I;
      );
      =     DB5.DBX 44.4;
NETWORK
TITLE =
      A     M 0.1;
      A(;
      A     DB5.DBX 6.6;
      A     M 0.2;
      O     DB5.DBX 4.2;
      O     DB1.DBX 0.5;
      );
      =     DB5.DBX 7.0;
NETWORK
TITLE =
      A     M 0.1;
      A(;
      A     DB5.DBX 9.0;
      A(;
      A     DB5.DBX 9.1;
      A     DB8.DBX 83.3;
      O;
      A     DB5.DBX 9.2;
      A(;
      O     DB5.DBX 3.3;
      O     DB5.DBX 6.5;
      );
      );
      O;
      A     DB5.DBX 9.3;
      A     DB2.DBX 26.0;
      A     DB5.DBX 3.3;
      );
      AN    DB5.DBX 44.5;
      =     L 0.0;
      A     L 0.0;
      BLD   102;
      =     DB5.DBX 6.5;
      A     L 0.0;
      FP    DB5.DBX 44.7;
      JNB   M023;
      L     0;
      T     DB5.DBW 50;
M023: NOP   0;
      A(;
      A     L 0.0;
      FN    M 800.5;
      );
      A     DB5.DBX 9.1;
      A     DB8.DBX 83.3;
      S     DB8.DBX 84.7;
NETWORK
TITLE =
      A     M 0.1;
      A     DB5.DBX 4.1;
      =     L 0.0;
      A     L 0.0;
      AN    DB5.DBX 44.5;
      A     M 0.3;
      JNB   M024;
      L     1;
      L     DB5.DBW 50;
      +I;
      T     DB5.DBW 50;
M024: NOP   0;
      A     L 0.0;
      A(;
      L     DB5.DBW 50;
      L     DB5.DBW 52;
      >=I;
      );
      =     DB5.DBX 44.5;
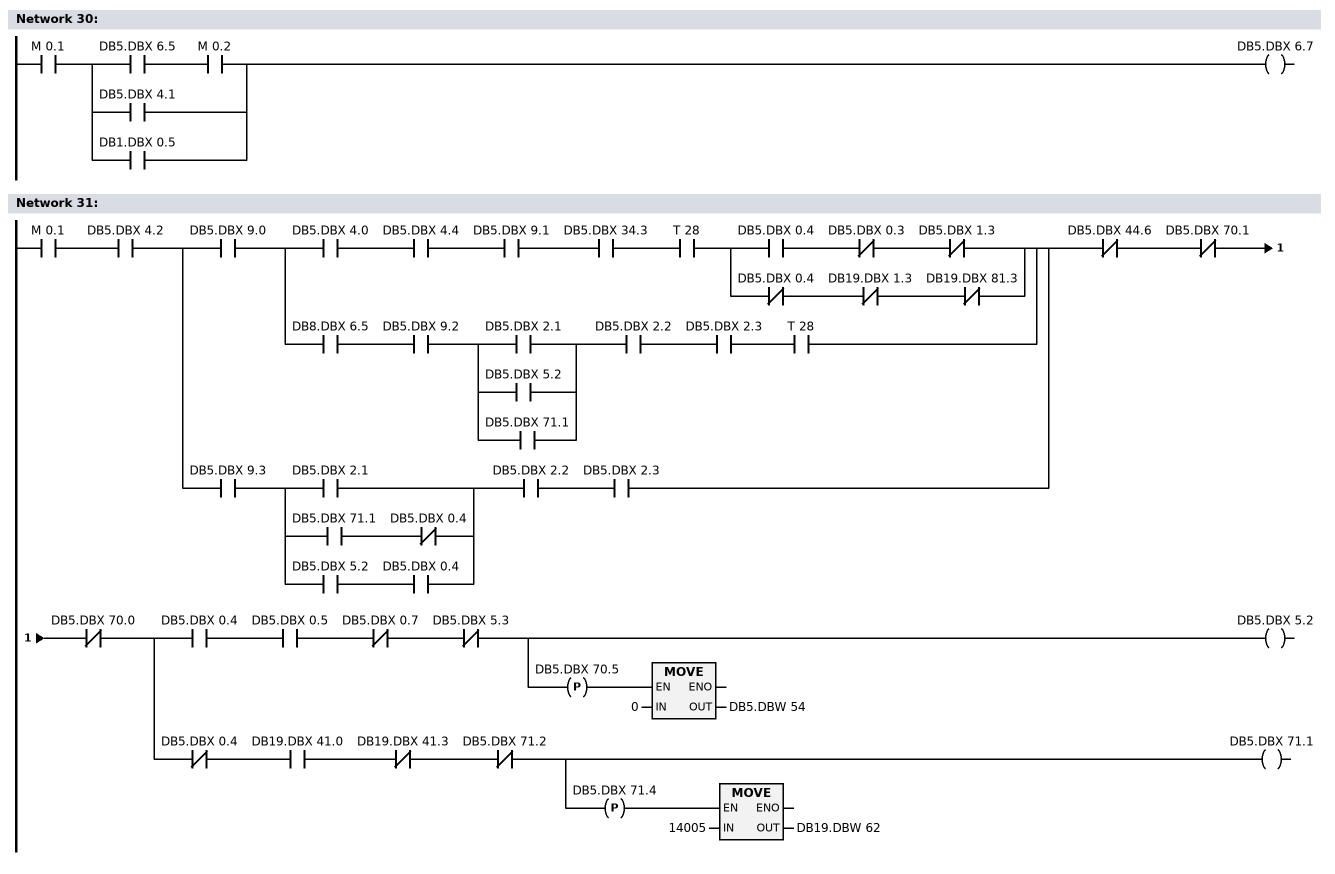
NETWORK
TITLE =
      A     M 0.1;
      A(;
      A     DB5.DBX 6.5;
      A     M 0.2;
      O     DB5.DBX 4.1;
      O     DB1.DBX 0.5;
      );
      =     DB5.DBX 6.7;
NETWORK
TITLE =
      A     M 0.1;
      A     DB5.DBX 4.2;
      A(;
      A     DB5.DBX 9.0;
      A(;
      A     DB5.DBX 4.0;
      A     DB5.DBX 4.4;
      A     DB5.DBX 9.1;
      A     DB5.DBX 34.3;
      A     T 28;
      A(;
      A     DB5.DBX 0.4;
      AN    DB5.DBX 0.3;
      AN    DB5.DBX 1.3;
      O;
      AN    DB5.DBX 0.4;
      AN    DB19.DBX 1.3;
      AN    DB19.DBX 81.3;
      );
      O;
      A     DB8.DBX 6.5;
      A     DB5.DBX 9.2;
      A(;
      O     DB5.DBX 2.1;
      O     DB5.DBX 5.2;
      O     DB5.DBX 71.1;
      );
      A     DB5.DBX 2.2;
      A     DB5.DBX 2.3;
      A     T 28;
      );
      O;
      A     DB5.DBX 9.3;
      A(;
      O     DB5.DBX 2.1;
      O;
      A     DB5.DBX 71.1;
      AN    DB5.DBX 0.4;
      O;
      A     DB5.DBX 5.2;
      A     DB5.DBX 0.4;
      );
      A     DB5.DBX 2.2;
      A     DB5.DBX 2.3;
      );
      AN    DB5.DBX 44.6;
      AN    DB5.DBX 70.1;
      AN    DB5.DBX 70.0;
      =     L 0.0;
      A     L 0.0;
      A     DB5.DBX 0.4;
      A     DB5.DBX 0.5;
      AN    DB5.DBX 0.7;
      AN    DB5.DBX 5.3;
      =     L 0.1;
      A     L 0.1;
      BLD   102;
      =     DB5.DBX 5.2;
      A     L 0.1;
      FP    DB5.DBX 70.5;
      JNB   M025;
      L     0;
      T     DB5.DBW 54;
M025: NOP   0;
      A     L 0.0;
      AN    DB5.DBX 0.4;
      A     DB19.DBX 41.0;
      AN    DB19.DBX 41.3;
      AN    DB5.DBX 71.2;
      =     L 0.1;
      A     L 0.1;
      BLD   102;
      =     DB5.DBX 71.1;
      A     L 0.1;
      FP    DB5.DBX 71.4;
      JNB   M026;
      L     14005;
      T     DB19.DBW 62;
M026: NOP   0;
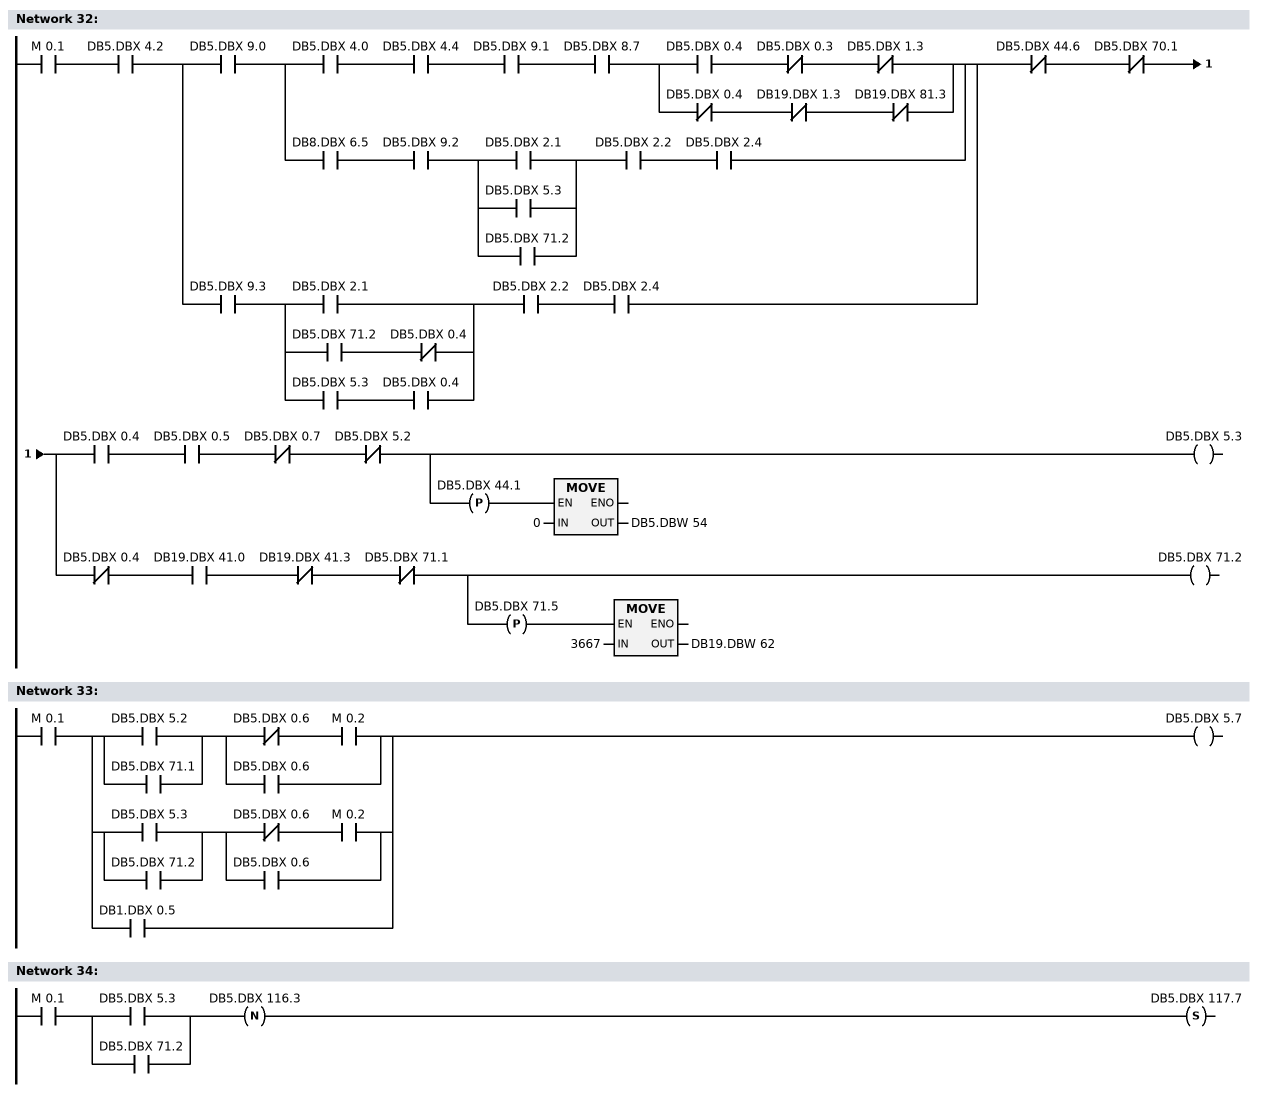
NETWORK
TITLE =
      A     M 0.1;
      A     DB5.DBX 4.2;
      A(;
      A     DB5.DBX 9.0;
      A(;
      A     DB5.DBX 4.0;
      A     DB5.DBX 4.4;
      A     DB5.DBX 9.1;
      A     DB5.DBX 8.7;
      A(;
      A     DB5.DBX 0.4;
      AN    DB5.DBX 0.3;
      AN    DB5.DBX 1.3;
      O;
      AN    DB5.DBX 0.4;
      AN    DB19.DBX 1.3;
      AN    DB19.DBX 81.3;
      );
      O;
      A     DB8.DBX 6.5;
      A     DB5.DBX 9.2;
      A(;
      O     DB5.DBX 2.1;
      O     DB5.DBX 5.3;
      O     DB5.DBX 71.2;
      );
      A     DB5.DBX 2.2;
      A     DB5.DBX 2.4;
      );
      O;
      A     DB5.DBX 9.3;
      A(;
      O     DB5.DBX 2.1;
      O;
      A     DB5.DBX 71.2;
      AN    DB5.DBX 0.4;
      O;
      A     DB5.DBX 5.3;
      A     DB5.DBX 0.4;
      );
      A     DB5.DBX 2.2;
      A     DB5.DBX 2.4;
      );
      AN    DB5.DBX 44.6;
      AN    DB5.DBX 70.1;
      =     L 0.0;
      A     L 0.0;
      A     DB5.DBX 0.4;
      A     DB5.DBX 0.5;
      AN    DB5.DBX 0.7;
      AN    DB5.DBX 5.2;
      =     L 0.1;
      A     L 0.1;
      BLD   102;
      =     DB5.DBX 5.3;
      A     L 0.1;
      FP    DB5.DBX 44.1;
      JNB   M027;
      L     0;
      T     DB5.DBW 54;
M027: NOP   0;
      A     L 0.0;
      AN    DB5.DBX 0.4;
      A     DB19.DBX 41.0;
      AN    DB19.DBX 41.3;
      AN    DB5.DBX 71.1;
      =     L 0.1;
      A     L 0.1;
      BLD   102;
      =     DB5.DBX 71.2;
      A     L 0.1;
      FP    DB5.DBX 71.5;
      JNB   M028;
      L     3667;
      T     DB19.DBW 62;
M028: NOP   0;
NETWORK
TITLE =
      A     M 0.1;
      A(;
      A(;
      O     DB5.DBX 5.2;
      O     DB5.DBX 71.1;
      );
      A(;
      AN    DB5.DBX 0.6;
      A     M 0.2;
      O     DB5.DBX 0.6;
      );
      O;
      A(;
      O     DB5.DBX 5.3;
      O     DB5.DBX 71.2;
      );
      A(;
      AN    DB5.DBX 0.6;
      A     M 0.2;
      O     DB5.DBX 0.6;
      );
      O     DB1.DBX 0.5;
      );
      =     DB5.DBX 5.7;
NETWORK
TITLE =
      A     M 0.1;
      A(;
      O     DB5.DBX 5.3;
      O     DB5.DBX 71.2;
      );
      FN    DB5.DBX 116.3;
      S     DB5.DBX 117.7;
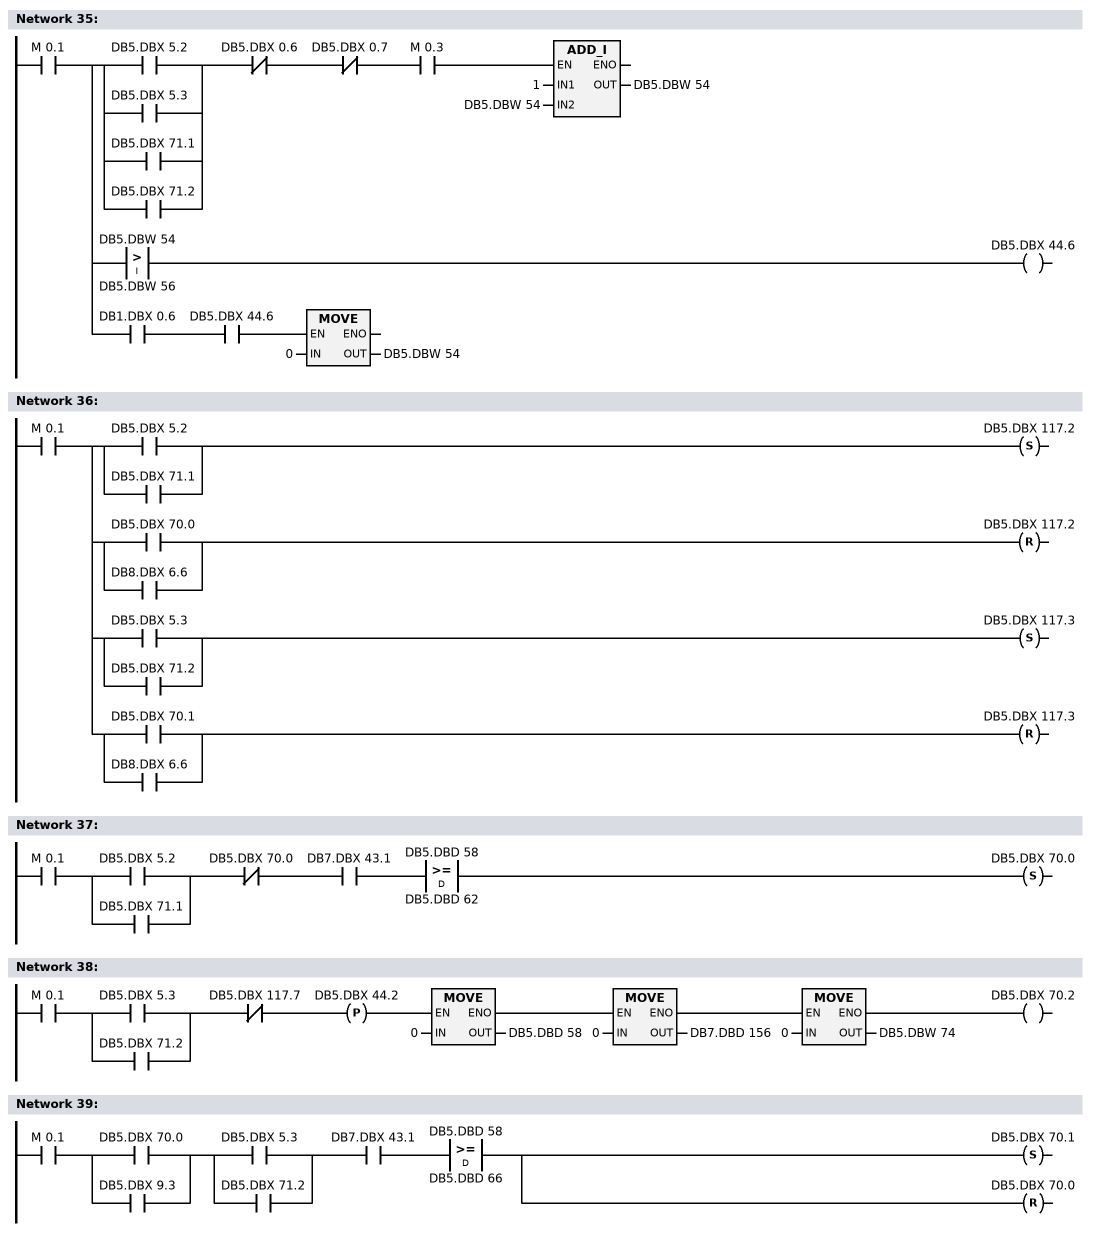
NETWORK
TITLE =
      A     M 0.1;
      =     L 0.0;
      A     L 0.0;
      A(;
      O     DB5.DBX 5.2;
      O     DB5.DBX 5.3;
      O     DB5.DBX 71.1;
      O     DB5.DBX 71.2;
      );
      AN    DB5.DBX 0.6;
      AN    DB5.DBX 0.7;
      A     M 0.3;
      JNB   M029;
      L     1;
      L     DB5.DBW 54;
      +I;
      T     DB5.DBW 54;
M029: NOP   0;
      A     L 0.0;
      A(;
      L     DB5.DBW 54;
      L     DB5.DBW 56;
      >I;
      );
      =     DB5.DBX 44.6;
      A     L 0.0;
      A     DB1.DBX 0.6;
      A     DB5.DBX 44.6;
      JNB   M030;
      L     0;
      T     DB5.DBW 54;
M030: NOP   0;
NETWORK
TITLE =
      A     M 0.1;
      =     L 0.0;
      A     L 0.0;
      A(;
      O     DB5.DBX 5.2;
      O     DB5.DBX 71.1;
      );
      S     DB5.DBX 117.2;
      A     L 0.0;
      A(;
      O     DB5.DBX 70.0;
      O     DB8.DBX 6.6;
      );
      R     DB5.DBX 117.2;
      A     L 0.0;
      A(;
      O     DB5.DBX 5.3;
      O     DB5.DBX 71.2;
      );
      S     DB5.DBX 117.3;
      A     L 0.0;
      A(;
      O     DB5.DBX 70.1;
      O     DB8.DBX 6.6;
      );
      R     DB5.DBX 117.3;
NETWORK
TITLE =
      A     M 0.1;
      A(;
      O     DB5.DBX 5.2;
      O     DB5.DBX 71.1;
      );
      AN    DB5.DBX 70.0;
      A     DB7.DBX 43.1;
      A(;
      L     DB5.DBD 58;
      L     DB5.DBD 62;
      >=D;
      );
      S     DB5.DBX 70.0;
NETWORK
TITLE =
      A(;
      A(;
      A     M 0.1;
      A(;
      O     DB5.DBX 5.3;
      O     DB5.DBX 71.2;
      );
      AN    DB5.DBX 117.7;
      FP    DB5.DBX 44.2;
      JNB   M031;
      L     0;
      T     DB5.DBD 58;
      SET;
      SAVE;
      CLR;
M031: A     BR;
      );
      JNB   M032;
      L     0;
      T     DB7.DBD 156;
      SET;
      SAVE;
      CLR;
M032: A     BR;
      );
      JNB   M033;
      L     0;
      T     DB5.DBW 74;
      SET;
      SAVE;
      CLR;
M033: A     BR;
      =     DB5.DBX 70.2;
NETWORK
TITLE =
      A     M 0.1;
      A(;
      O     DB5.DBX 70.0;
      O     DB5.DBX 9.3;
      );
      A(;
      O     DB5.DBX 5.3;
      O     DB5.DBX 71.2;
      );
      A     DB7.DBX 43.1;
      A(;
      L     DB5.DBD 58;
      L     DB5.DBD 66;
      >=D;
      );
      S     DB5.DBX 70.1;
      R     DB5.DBX 70.0;
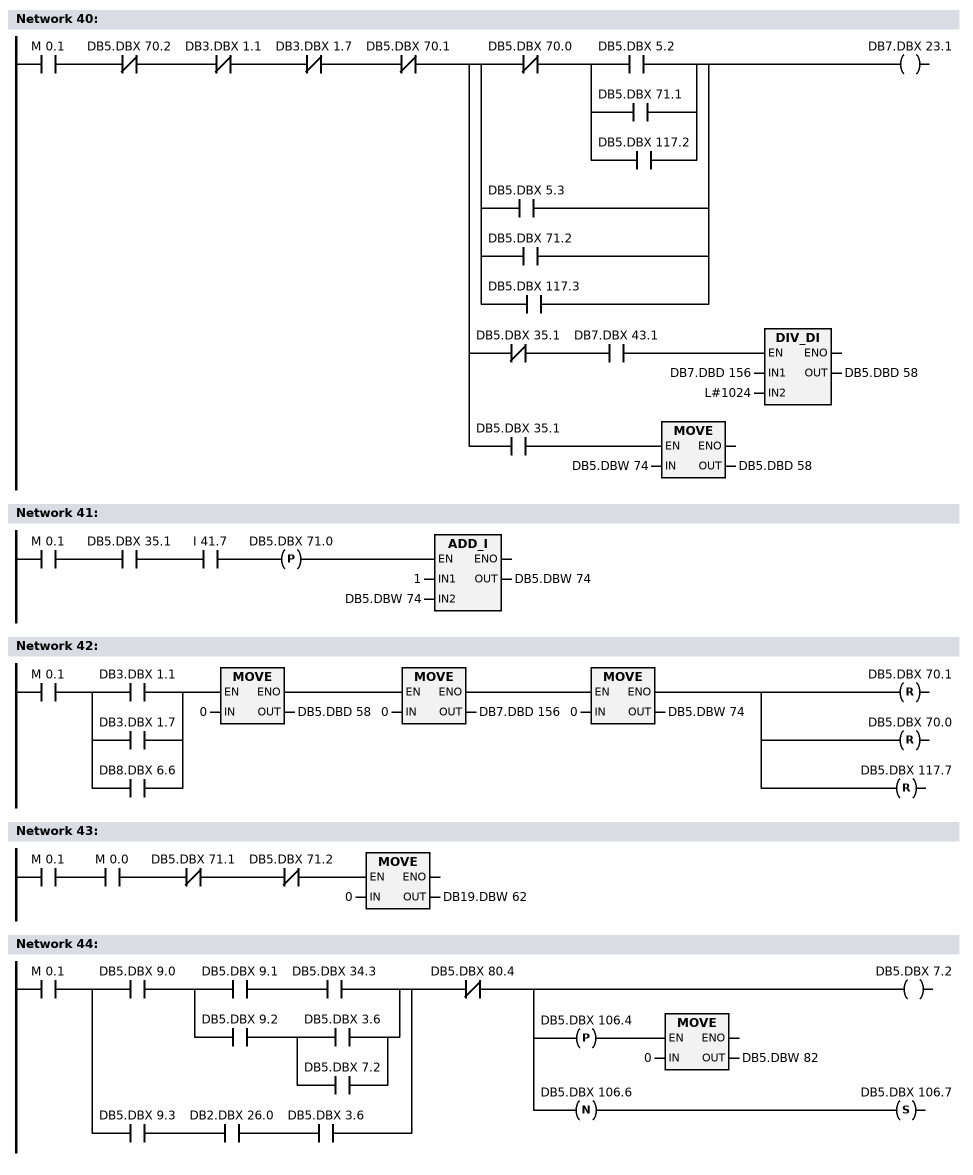
NETWORK
TITLE =
      A     M 0.1;
      AN    DB5.DBX 70.2;
      AN    DB3.DBX 1.1;
      AN    DB3.DBX 1.7;
      AN    DB5.DBX 70.1;
      =     L 0.0;
      A     L 0.0;
      A(;
      AN    DB5.DBX 70.0;
      A(;
      O     DB5.DBX 5.2;
      O     DB5.DBX 71.1;
      O     DB5.DBX 117.2;
      );
      O     DB5.DBX 5.3;
      O     DB5.DBX 71.2;
      O     DB5.DBX 117.3;
      );
      =     DB7.DBX 23.1;
      A     L 0.0;
      AN    DB5.DBX 35.1;
      A     DB7.DBX 43.1;
      JNB   M034;
      L     DB7.DBD 156;
      L     L#1024;
      /D;
      T     DB5.DBD 58;
M034: NOP   0;
      A     L 0.0;
      A     DB5.DBX 35.1;
      JNB   M035;
      L     DB5.DBW 74;
      T     DB5.DBD 58;
M035: NOP   0;
NETWORK
TITLE =
      A     M 0.1;
      A     DB5.DBX 35.1;
      A     I 41.7;
      FP    DB5.DBX 71.0;
      JNB   M036;
      L     1;
      L     DB5.DBW 74;
      +I;
      T     DB5.DBW 74;
M036: NOP   0;
NETWORK
TITLE =
      A(;
      A(;
      A     M 0.1;
      A(;
      O     DB3.DBX 1.1;
      O     DB3.DBX 1.7;
      O     DB8.DBX 6.6;
      );
      JNB   M037;
      L     0;
      T     DB5.DBD 58;
      SET;
      SAVE;
      CLR;
M037: A     BR;
      );
      JNB   M038;
      L     0;
      T     DB7.DBD 156;
      SET;
      SAVE;
      CLR;
M038: A     BR;
      );
      JNB   M039;
      L     0;
      T     DB5.DBW 74;
      SET;
      SAVE;
      CLR;
M039: A     BR;
      R     DB5.DBX 70.1;
      R     DB5.DBX 70.0;
      R     DB5.DBX 117.7;
NETWORK
TITLE =
      A     M 0.1;
      A     M 0.0;
      AN    DB5.DBX 71.1;
      AN    DB5.DBX 71.2;
      JNB   M040;
      L     0;
      T     DB19.DBW 62;
M040: NOP   0;
NETWORK
TITLE =
      A     M 0.1;
      A(;
      A     DB5.DBX 9.0;
      A(;
      A     DB5.DBX 9.1;
      A     DB5.DBX 34.3;
      O;
      A     DB5.DBX 9.2;
      A(;
      O     DB5.DBX 3.6;
      O     DB5.DBX 7.2;
      );
      );
      O;
      A     DB5.DBX 9.3;
      A     DB2.DBX 26.0;
      A     DB5.DBX 3.6;
      );
      AN    DB5.DBX 80.4;
      =     L 0.0;
      A     L 0.0;
      BLD   102;
      =     DB5.DBX 7.2;
      A     L 0.0;
      FP    DB5.DBX 106.4;
      JNB   M041;
      L     0;
      T     DB5.DBW 82;
M041: NOP   0;
      A     L 0.0;
      FN    DB5.DBX 106.6;
      S     DB5.DBX 106.7;
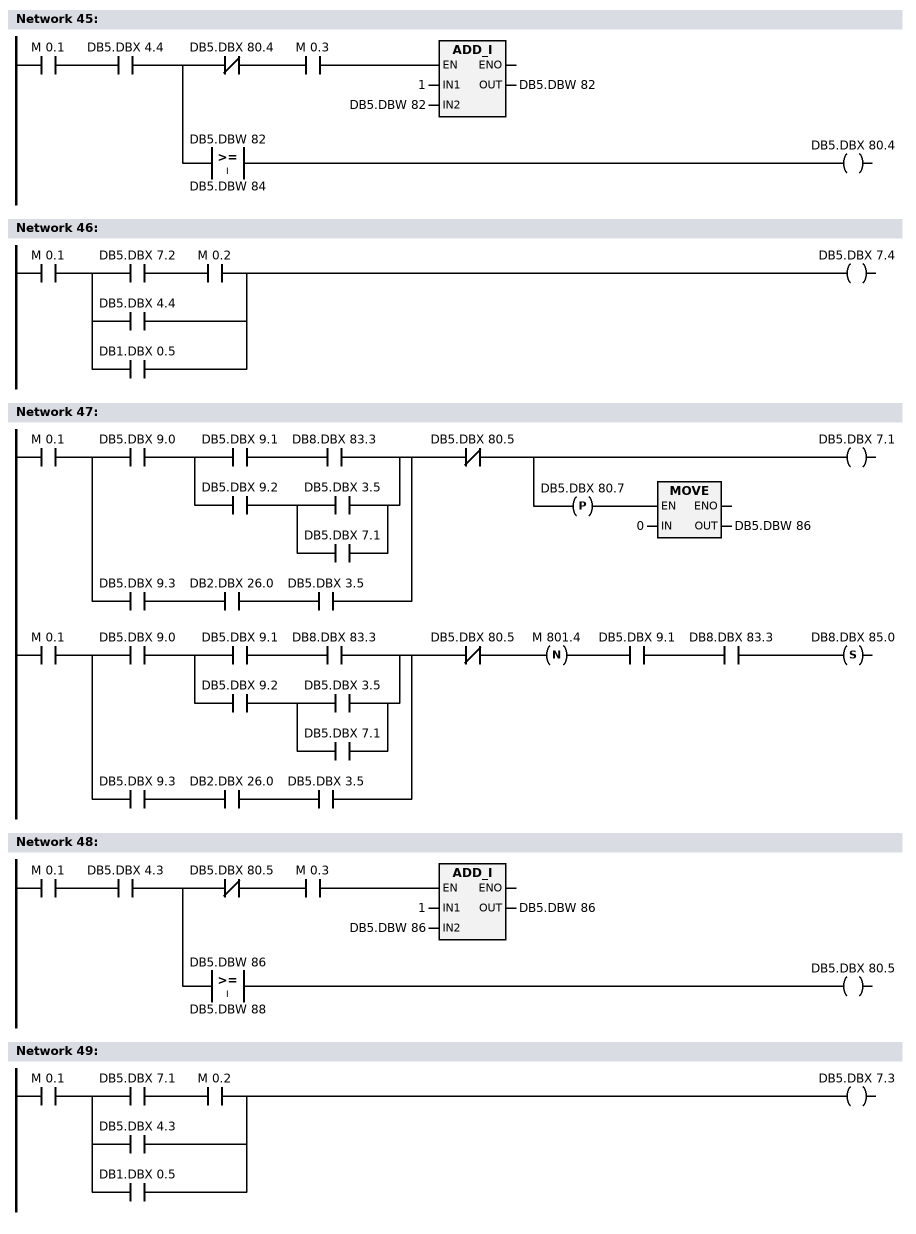
NETWORK
TITLE =
      A     M 0.1;
      A     DB5.DBX 4.4;
      =     L 0.0;
      A     L 0.0;
      AN    DB5.DBX 80.4;
      A     M 0.3;
      JNB   M042;
      L     1;
      L     DB5.DBW 82;
      +I;
      T     DB5.DBW 82;
M042: NOP   0;
      A     L 0.0;
      A(;
      L     DB5.DBW 82;
      L     DB5.DBW 84;
      >=I;
      );
      =     DB5.DBX 80.4;
NETWORK
TITLE =
      A     M 0.1;
      A(;
      A     DB5.DBX 7.2;
      A     M 0.2;
      O     DB5.DBX 4.4;
      O     DB1.DBX 0.5;
      );
      =     DB5.DBX 7.4;
NETWORK
TITLE =
      A     M 0.1;
      A(;
      A     DB5.DBX 9.0;
      A(;
      A     DB5.DBX 9.1;
      A     DB8.DBX 83.3;
      O;
      A     DB5.DBX 9.2;
      A(;
      O     DB5.DBX 3.5;
      O     DB5.DBX 7.1;
      );
      );
      O;
      A     DB5.DBX 9.3;
      A     DB2.DBX 26.0;
      A     DB5.DBX 3.5;
      );
      AN    DB5.DBX 80.5;
      =     L 0.0;
      A     L 0.0;
      BLD   102;
      =     DB5.DBX 7.1;
      A     L 0.0;
      FP    DB5.DBX 80.7;
      JNB   M043;
      L     0;
      T     DB5.DBW 86;
M043: NOP   0;
      A(;
      A     L 0.0;
      FN    M 801.4;
      );
      A     DB5.DBX 9.1;
      A     DB8.DBX 83.3;
      S     DB8.DBX 85.0;
NETWORK
TITLE =
      A     M 0.1;
      A     DB5.DBX 4.3;
      =     L 0.0;
      A     L 0.0;
      AN    DB5.DBX 80.5;
      A     M 0.3;
      JNB   M044;
      L     1;
      L     DB5.DBW 86;
      +I;
      T     DB5.DBW 86;
M044: NOP   0;
      A     L 0.0;
      A(;
      L     DB5.DBW 86;
      L     DB5.DBW 88;
      >=I;
      );
      =     DB5.DBX 80.5;
NETWORK
TITLE =
      A     M 0.1;
      A(;
      A     DB5.DBX 7.1;
      A     M 0.2;
      O     DB5.DBX 4.3;
      O     DB1.DBX 0.5;
      );
      =     DB5.DBX 7.3;
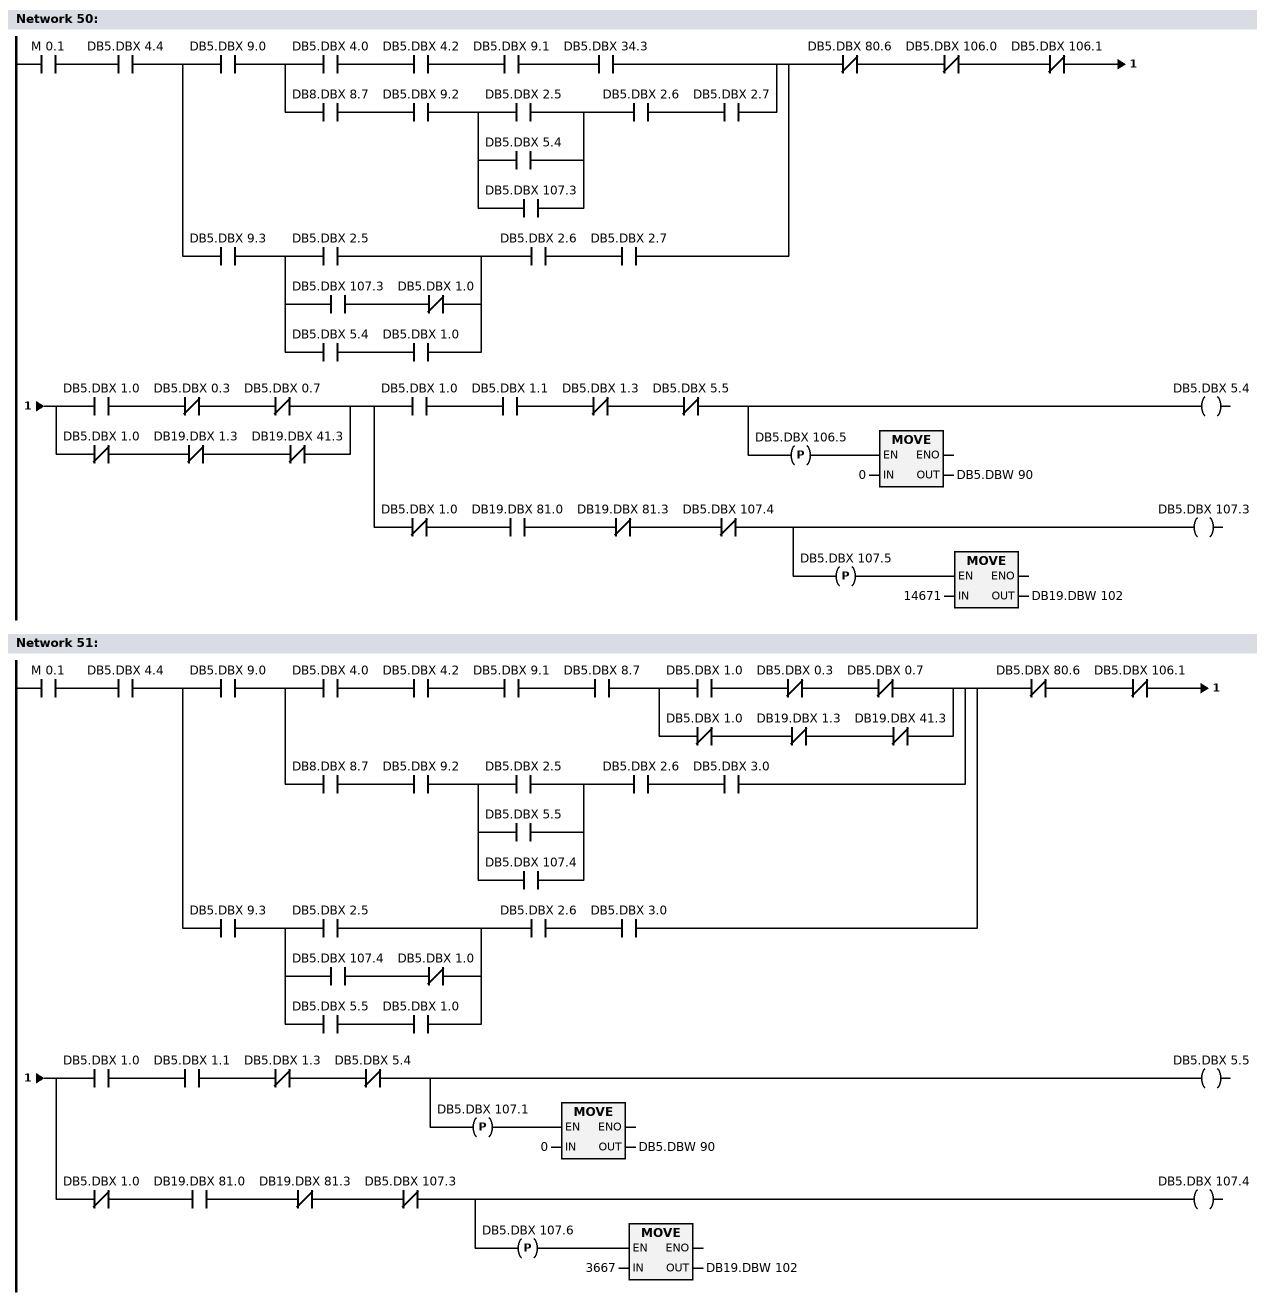
NETWORK
TITLE =
      A     M 0.1;
      A     DB5.DBX 4.4;
      A(;
      A     DB5.DBX 9.0;
      A(;
      A     DB5.DBX 4.0;
      A     DB5.DBX 4.2;
      A     DB5.DBX 9.1;
      A     DB5.DBX 34.3;
      O;
      A     DB8.DBX 8.7;
      A     DB5.DBX 9.2;
      A(;
      O     DB5.DBX 2.5;
      O     DB5.DBX 5.4;
      O     DB5.DBX 107.3;
      );
      A     DB5.DBX 2.6;
      A     DB5.DBX 2.7;
      );
      O;
      A     DB5.DBX 9.3;
      A(;
      O     DB5.DBX 2.5;
      O;
      A     DB5.DBX 107.3;
      AN    DB5.DBX 1.0;
      O;
      A     DB5.DBX 5.4;
      A     DB5.DBX 1.0;
      );
      A     DB5.DBX 2.6;
      A     DB5.DBX 2.7;
      );
      AN    DB5.DBX 80.6;
      AN    DB5.DBX 106.0;
      AN    DB5.DBX 106.1;
      A(;
      A     DB5.DBX 1.0;
      AN    DB5.DBX 0.3;
      AN    DB5.DBX 0.7;
      O;
      AN    DB5.DBX 1.0;
      AN    DB19.DBX 1.3;
      AN    DB19.DBX 41.3;
      );
      =     L 0.0;
      A     L 0.0;
      A     DB5.DBX 1.0;
      A     DB5.DBX 1.1;
      AN    DB5.DBX 1.3;
      AN    DB5.DBX 5.5;
      =     L 0.1;
      A     L 0.1;
      BLD   102;
      =     DB5.DBX 5.4;
      A     L 0.1;
      FP    DB5.DBX 106.5;
      JNB   M045;
      L     0;
      T     DB5.DBW 90;
M045: NOP   0;
      A     L 0.0;
      AN    DB5.DBX 1.0;
      A     DB19.DBX 81.0;
      AN    DB19.DBX 81.3;
      AN    DB5.DBX 107.4;
      =     L 0.1;
      A     L 0.1;
      BLD   102;
      =     DB5.DBX 107.3;
      A     L 0.1;
      FP    DB5.DBX 107.5;
      JNB   M046;
      L     14671;
      T     DB19.DBW 102;
M046: NOP   0;
NETWORK
TITLE =
      A     M 0.1;
      A     DB5.DBX 4.4;
      A(;
      A     DB5.DBX 9.0;
      A(;
      A     DB5.DBX 4.0;
      A     DB5.DBX 4.2;
      A     DB5.DBX 9.1;
      A     DB5.DBX 8.7;
      A(;
      A     DB5.DBX 1.0;
      AN    DB5.DBX 0.3;
      AN    DB5.DBX 0.7;
      O;
      AN    DB5.DBX 1.0;
      AN    DB19.DBX 1.3;
      AN    DB19.DBX 41.3;
      );
      O;
      A     DB8.DBX 8.7;
      A     DB5.DBX 9.2;
      A(;
      O     DB5.DBX 2.5;
      O     DB5.DBX 5.5;
      O     DB5.DBX 107.4;
      );
      A     DB5.DBX 2.6;
      A     DB5.DBX 3.0;
      );
      O;
      A     DB5.DBX 9.3;
      A(;
      O     DB5.DBX 2.5;
      O;
      A     DB5.DBX 107.4;
      AN    DB5.DBX 1.0;
      O;
      A     DB5.DBX 5.5;
      A     DB5.DBX 1.0;
      );
      A     DB5.DBX 2.6;
      A     DB5.DBX 3.0;
      );
      AN    DB5.DBX 80.6;
      AN    DB5.DBX 106.1;
      =     L 0.0;
      A     L 0.0;
      A     DB5.DBX 1.0;
      A     DB5.DBX 1.1;
      AN    DB5.DBX 1.3;
      AN    DB5.DBX 5.4;
      =     L 0.1;
      A     L 0.1;
      BLD   102;
      =     DB5.DBX 5.5;
      A     L 0.1;
      FP    DB5.DBX 107.1;
      JNB   M047;
      L     0;
      T     DB5.DBW 90;
M047: NOP   0;
      A     L 0.0;
      AN    DB5.DBX 1.0;
      A     DB19.DBX 81.0;
      AN    DB19.DBX 81.3;
      AN    DB5.DBX 107.3;
      =     L 0.1;
      A     L 0.1;
      BLD   102;
      =     DB5.DBX 107.4;
      A     L 0.1;
      FP    DB5.DBX 107.6;
      JNB   M048;
      L     3667;
      T     DB19.DBW 102;
M048: NOP   0;
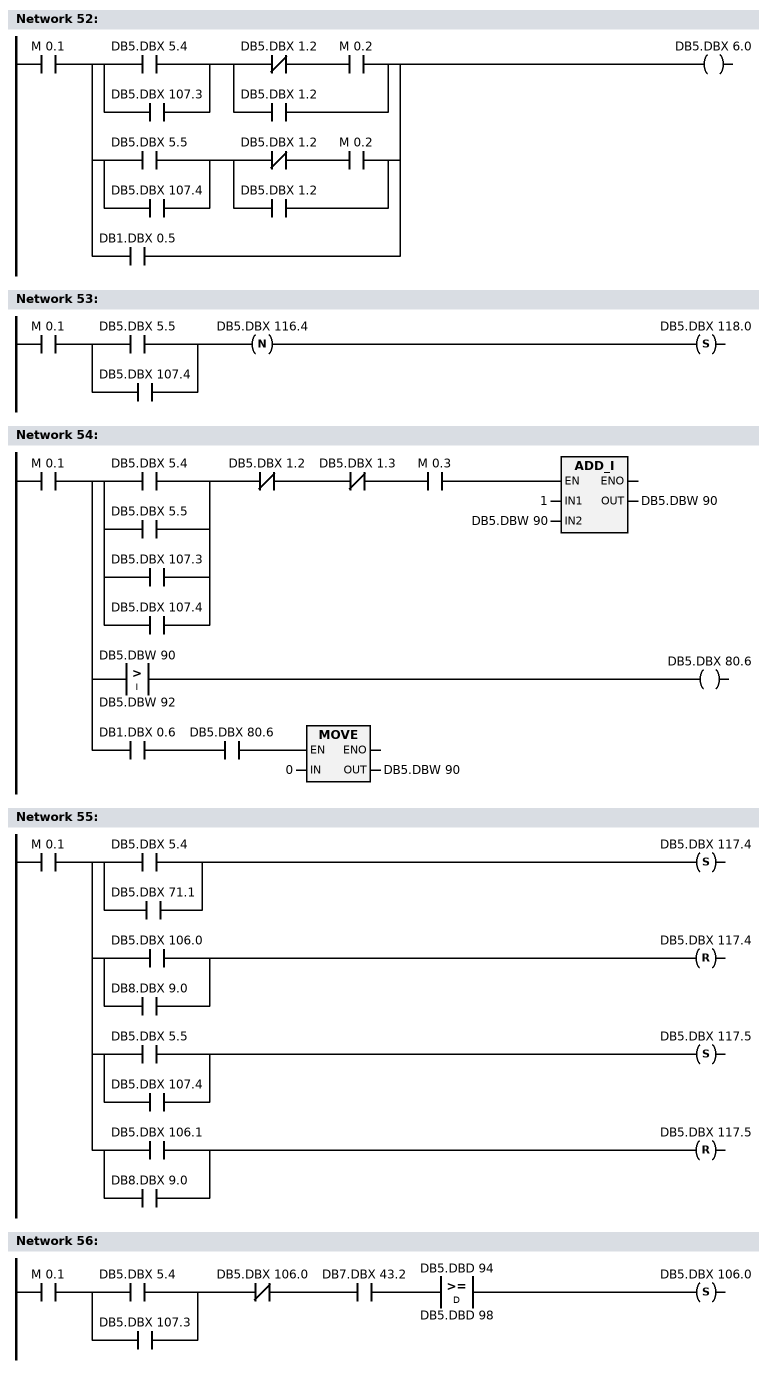
NETWORK
TITLE =
      A     M 0.1;
      A(;
      A(;
      O     DB5.DBX 5.4;
      O     DB5.DBX 107.3;
      );
      A(;
      AN    DB5.DBX 1.2;
      A     M 0.2;
      O     DB5.DBX 1.2;
      );
      O;
      A(;
      O     DB5.DBX 5.5;
      O     DB5.DBX 107.4;
      );
      A(;
      AN    DB5.DBX 1.2;
      A     M 0.2;
      O     DB5.DBX 1.2;
      );
      O     DB1.DBX 0.5;
      );
      =     DB5.DBX 6.0;
NETWORK
TITLE =
      A     M 0.1;
      A(;
      O     DB5.DBX 5.5;
      O     DB5.DBX 107.4;
      );
      FN    DB5.DBX 116.4;
      S     DB5.DBX 118.0;
NETWORK
TITLE =
      A     M 0.1;
      =     L 0.0;
      A     L 0.0;
      A(;
      O     DB5.DBX 5.4;
      O     DB5.DBX 5.5;
      O     DB5.DBX 107.3;
      O     DB5.DBX 107.4;
      );
      AN    DB5.DBX 1.2;
      AN    DB5.DBX 1.3;
      A     M 0.3;
      JNB   M049;
      L     1;
      L     DB5.DBW 90;
      +I;
      T     DB5.DBW 90;
M049: NOP   0;
      A     L 0.0;
      A(;
      L     DB5.DBW 90;
      L     DB5.DBW 92;
      >I;
      );
      =     DB5.DBX 80.6;
      A     L 0.0;
      A     DB1.DBX 0.6;
      A     DB5.DBX 80.6;
      JNB   M050;
      L     0;
      T     DB5.DBW 90;
M050: NOP   0;
NETWORK
TITLE =
      A     M 0.1;
      =     L 0.0;
      A     L 0.0;
      A(;
      O     DB5.DBX 5.4;
      O     DB5.DBX 71.1;
      );
      S     DB5.DBX 117.4;
      A     L 0.0;
      A(;
      O     DB5.DBX 106.0;
      O     DB8.DBX 9.0;
      );
      R     DB5.DBX 117.4;
      A     L 0.0;
      A(;
      O     DB5.DBX 5.5;
      O     DB5.DBX 107.4;
      );
      S     DB5.DBX 117.5;
      A     L 0.0;
      A(;
      O     DB5.DBX 106.1;
      O     DB8.DBX 9.0;
      );
      R     DB5.DBX 117.5;
NETWORK
TITLE =
      A     M 0.1;
      A(;
      O     DB5.DBX 5.4;
      O     DB5.DBX 107.3;
      );
      AN    DB5.DBX 106.0;
      A     DB7.DBX 43.2;
      A(;
      L     DB5.DBD 94;
      L     DB5.DBD 98;
      >=D;
      );
      S     DB5.DBX 106.0;
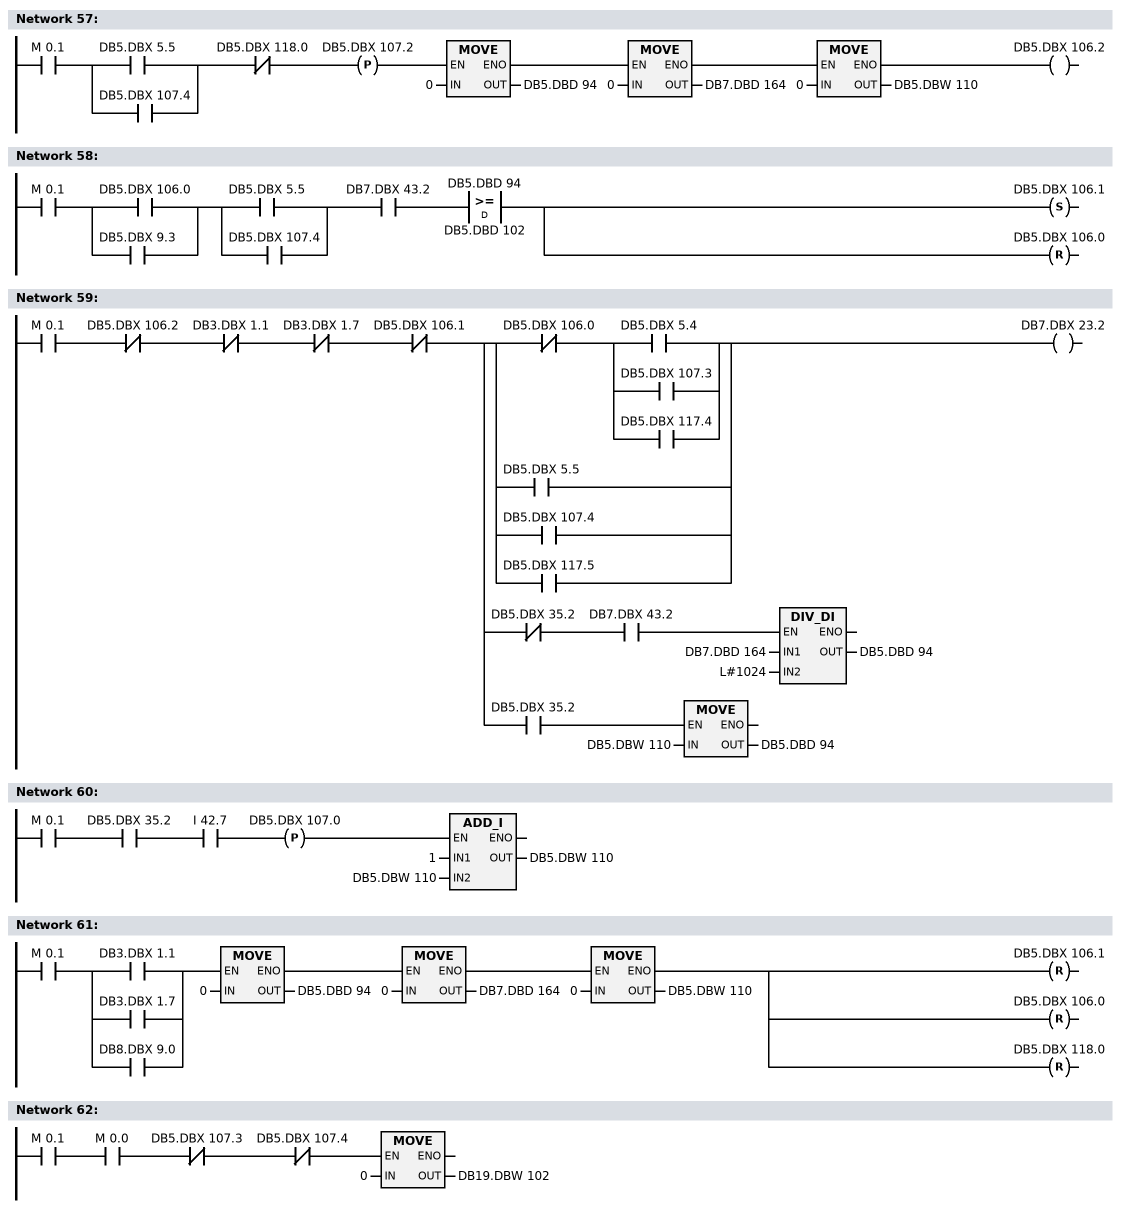
NETWORK
TITLE =
      A(;
      A(;
      A     M 0.1;
      A(;
      O     DB5.DBX 5.5;
      O     DB5.DBX 107.4;
      );
      AN    DB5.DBX 118.0;
      FP    DB5.DBX 107.2;
      JNB   M051;
      L     0;
      T     DB5.DBD 94;
      SET;
      SAVE;
      CLR;
M051: A     BR;
      );
      JNB   M052;
      L     0;
      T     DB7.DBD 164;
      SET;
      SAVE;
      CLR;
M052: A     BR;
      );
      JNB   M053;
      L     0;
      T     DB5.DBW 110;
      SET;
      SAVE;
      CLR;
M053: A     BR;
      =     DB5.DBX 106.2;
NETWORK
TITLE =
      A     M 0.1;
      A(;
      O     DB5.DBX 106.0;
      O     DB5.DBX 9.3;
      );
      A(;
      O     DB5.DBX 5.5;
      O     DB5.DBX 107.4;
      );
      A     DB7.DBX 43.2;
      A(;
      L     DB5.DBD 94;
      L     DB5.DBD 102;
      >=D;
      );
      S     DB5.DBX 106.1;
      R     DB5.DBX 106.0;
NETWORK
TITLE =
      A     M 0.1;
      AN    DB5.DBX 106.2;
      AN    DB3.DBX 1.1;
      AN    DB3.DBX 1.7;
      AN    DB5.DBX 106.1;
      =     L 0.0;
      A     L 0.0;
      A(;
      AN    DB5.DBX 106.0;
      A(;
      O     DB5.DBX 5.4;
      O     DB5.DBX 107.3;
      O     DB5.DBX 117.4;
      );
      O     DB5.DBX 5.5;
      O     DB5.DBX 107.4;
      O     DB5.DBX 117.5;
      );
      =     DB7.DBX 23.2;
      A     L 0.0;
      AN    DB5.DBX 35.2;
      A     DB7.DBX 43.2;
      JNB   M054;
      L     DB7.DBD 164;
      L     L#1024;
      /D;
      T     DB5.DBD 94;
M054: NOP   0;
      A     L 0.0;
      A     DB5.DBX 35.2;
      JNB   M055;
      L     DB5.DBW 110;
      T     DB5.DBD 94;
M055: NOP   0;
NETWORK
TITLE =
      A     M 0.1;
      A     DB5.DBX 35.2;
      A     I 42.7;
      FP    DB5.DBX 107.0;
      JNB   M056;
      L     1;
      L     DB5.DBW 110;
      +I;
      T     DB5.DBW 110;
M056: NOP   0;
NETWORK
TITLE =
      A(;
      A(;
      A     M 0.1;
      A(;
      O     DB3.DBX 1.1;
      O     DB3.DBX 1.7;
      O     DB8.DBX 9.0;
      );
      JNB   M057;
      L     0;
      T     DB5.DBD 94;
      SET;
      SAVE;
      CLR;
M057: A     BR;
      );
      JNB   M058;
      L     0;
      T     DB7.DBD 164;
      SET;
      SAVE;
      CLR;
M058: A     BR;
      );
      JNB   M059;
      L     0;
      T     DB5.DBW 110;
      SET;
      SAVE;
      CLR;
M059: A     BR;
      R     DB5.DBX 106.1;
      R     DB5.DBX 106.0;
      R     DB5.DBX 118.0;
NETWORK
TITLE =
      A     M 0.1;
      A     M 0.0;
      AN    DB5.DBX 107.3;
      AN    DB5.DBX 107.4;
      JNB   M060;
      L     0;
      T     DB19.DBW 102;
M060: NOP   0;
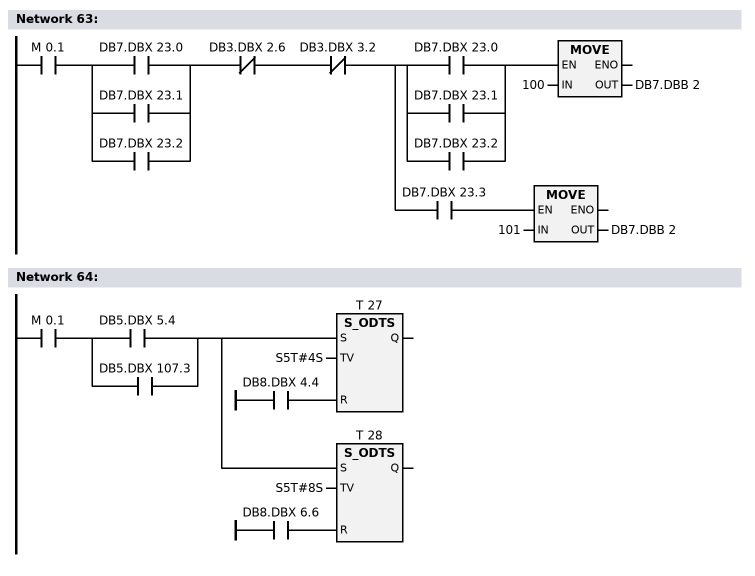
NETWORK
TITLE =
      A     M 0.1;
      A(;
      O     DB7.DBX 23.0;
      O     DB7.DBX 23.1;
      O     DB7.DBX 23.2;
      );
      AN    DB3.DBX 2.6;
      AN    DB3.DBX 3.2;
      =     L 0.0;
      A     L 0.0;
      A(;
      O     DB7.DBX 23.0;
      O     DB7.DBX 23.1;
      O     DB7.DBX 23.2;
      );
      JNB   M061;
      L     100;
      T     DB7.DBB 2;
M061: NOP   0;
      A     L 0.0;
      A     DB7.DBX 23.3;
      JNB   M062;
      L     101;
      T     DB7.DBB 2;
M062: NOP   0;
NETWORK
TITLE =
      A     M 0.1;
      A(;
      O     DB5.DBX 5.4;
      O     DB5.DBX 107.3;
      );
      =     L 0.0;
      A     L 0.0;
      L     S5T#4S;
      SS    T 27;
      A     DB8.DBX 4.4;
      R     T 27;
      NOP   0;
      NOP   0;
      NOP   0;
      A     L 0.0;
      L     S5T#8S;
      SS    T 28;
      A     DB8.DBX 6.6;
      R     T 28;
      NOP   0;
      NOP   0;
      NOP   0;
END_FUNCTION

FUNCTION FC 11 : VOID
AUTHOR : Arun
VERSION : 0.1
BEGIN
// (block stored without names or comments; labels and parameter names are numbered)
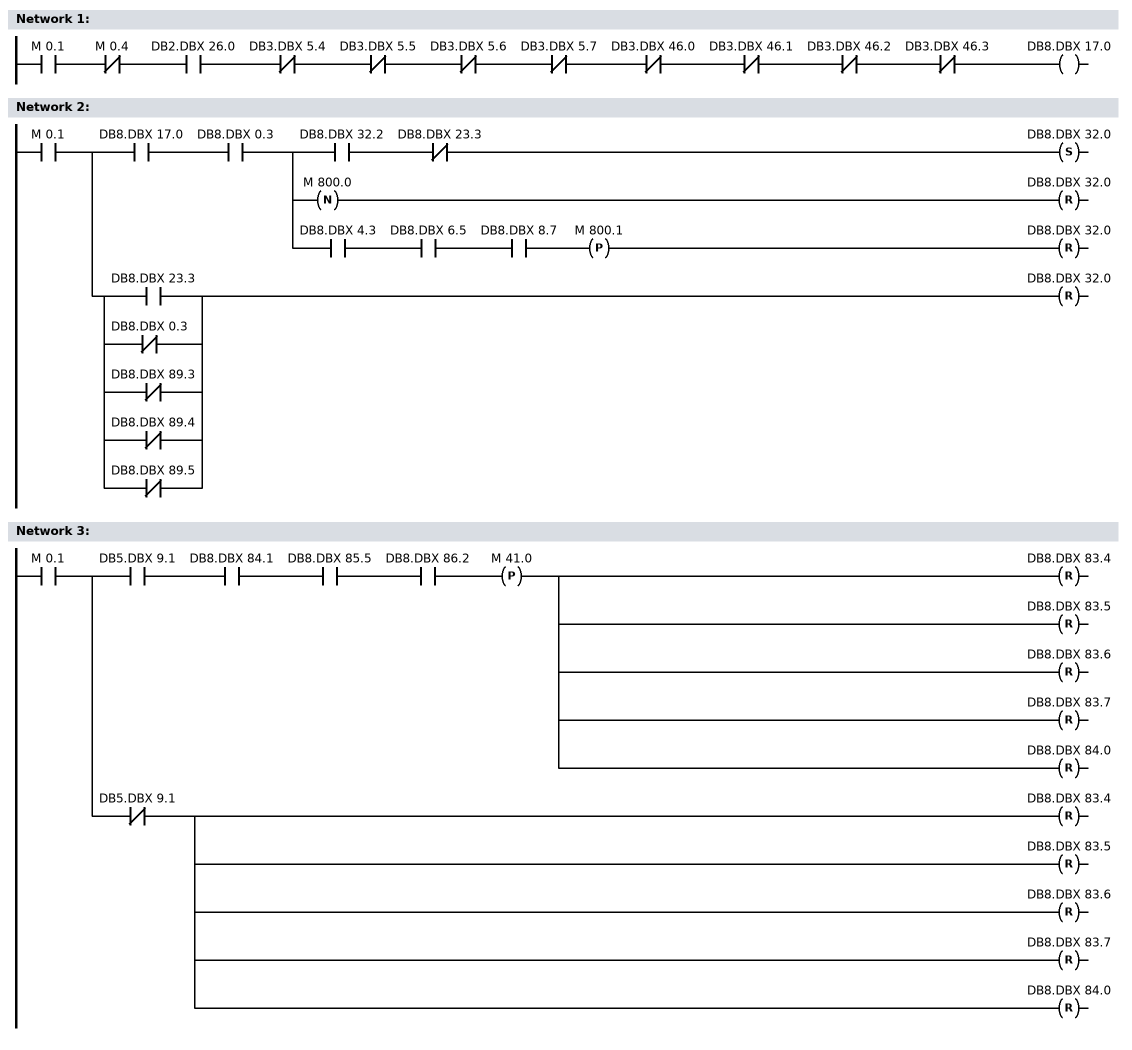
NETWORK
TITLE =
      A     M 0.1;
      AN    M 0.4;
      A     DB2.DBX 26.0;
      AN    DB3.DBX 5.4;
      AN    DB3.DBX 5.5;
      AN    DB3.DBX 5.6;
      AN    DB3.DBX 5.7;
      AN    DB3.DBX 46.0;
      AN    DB3.DBX 46.1;
      AN    DB3.DBX 46.2;
      AN    DB3.DBX 46.3;
      =     DB8.DBX 17.0;
NETWORK
TITLE =
      A     M 0.1;
      =     L 0.0;
      A     L 0.0;
      A     DB8.DBX 17.0;
      A     DB8.DBX 0.3;
      =     L 0.1;
      A     L 0.1;
      A     DB8.DBX 32.2;
      AN    DB8.DBX 23.3;
      S     DB8.DBX 32.0;
      A     L 0.1;
      FN    M 800.0;
      R     DB8.DBX 32.0;
      A     L 0.1;
      A     DB8.DBX 4.3;
      A     DB8.DBX 6.5;
      A     DB8.DBX 8.7;
      FP    M 800.1;
      R     DB8.DBX 32.0;
      A     L 0.0;
      A(;
      O     DB8.DBX 23.3;
      ON    DB8.DBX 0.3;
      ON    DB8.DBX 89.3;
      ON    DB8.DBX 89.4;
      ON    DB8.DBX 89.5;
      );
      R     DB8.DBX 32.0;
NETWORK
TITLE =
      A     M 0.1;
      =     L 0.0;
      A     L 0.0;
      A     DB5.DBX 9.1;
      A     DB8.DBX 84.1;
      A     DB8.DBX 85.5;
      A     DB8.DBX 86.2;
      FP    M 41.0;
      R     DB8.DBX 83.4;
      R     DB8.DBX 83.5;
      R     DB8.DBX 83.6;
      R     DB8.DBX 83.7;
      R     DB8.DBX 84.0;
      A     L 0.0;
      AN    DB5.DBX 9.1;
      R     DB8.DBX 83.4;
      R     DB8.DBX 83.5;
      R     DB8.DBX 83.6;
      R     DB8.DBX 83.7;
      R     DB8.DBX 84.0;
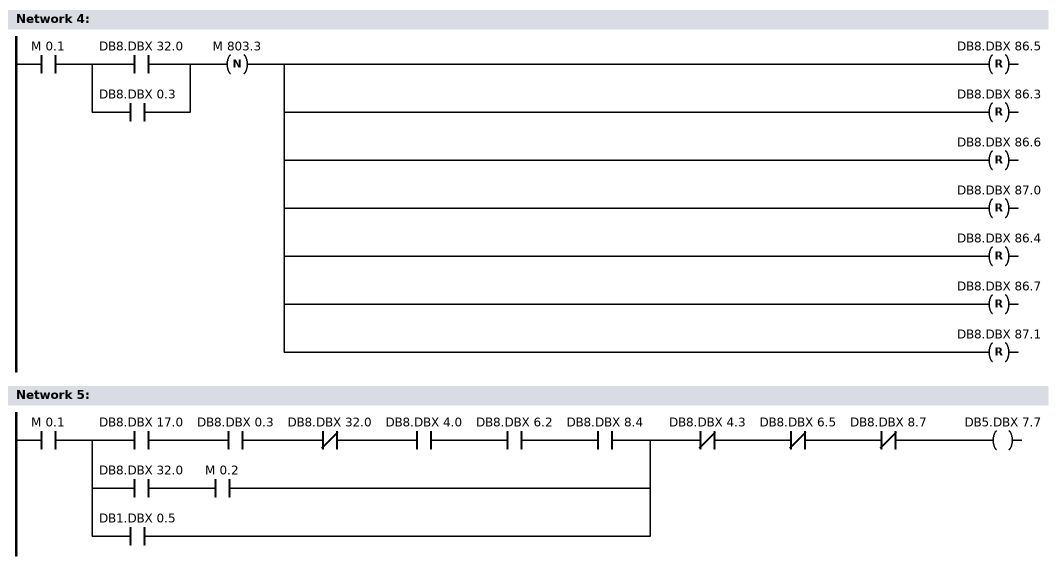
NETWORK
TITLE =
      A     M 0.1;
      A(;
      O     DB8.DBX 32.0;
      O     DB8.DBX 0.3;
      );
      FN    M 803.3;
      R     DB8.DBX 86.5;
      R     DB8.DBX 86.3;
      R     DB8.DBX 86.6;
      R     DB8.DBX 87.0;
      R     DB8.DBX 86.4;
      R     DB8.DBX 86.7;
      R     DB8.DBX 87.1;
NETWORK
TITLE =
      A     M 0.1;
      A(;
      A     DB8.DBX 17.0;
      A     DB8.DBX 0.3;
      AN    DB8.DBX 32.0;
      A     DB8.DBX 4.0;
      A     DB8.DBX 6.2;
      A     DB8.DBX 8.4;
      O;
      A     DB8.DBX 32.0;
      A     M 0.2;
      O     DB1.DBX 0.5;
      );
      AN    DB8.DBX 4.3;
      AN    DB8.DBX 6.5;
      AN    DB8.DBX 8.7;
      =     DB5.DBX 7.7;
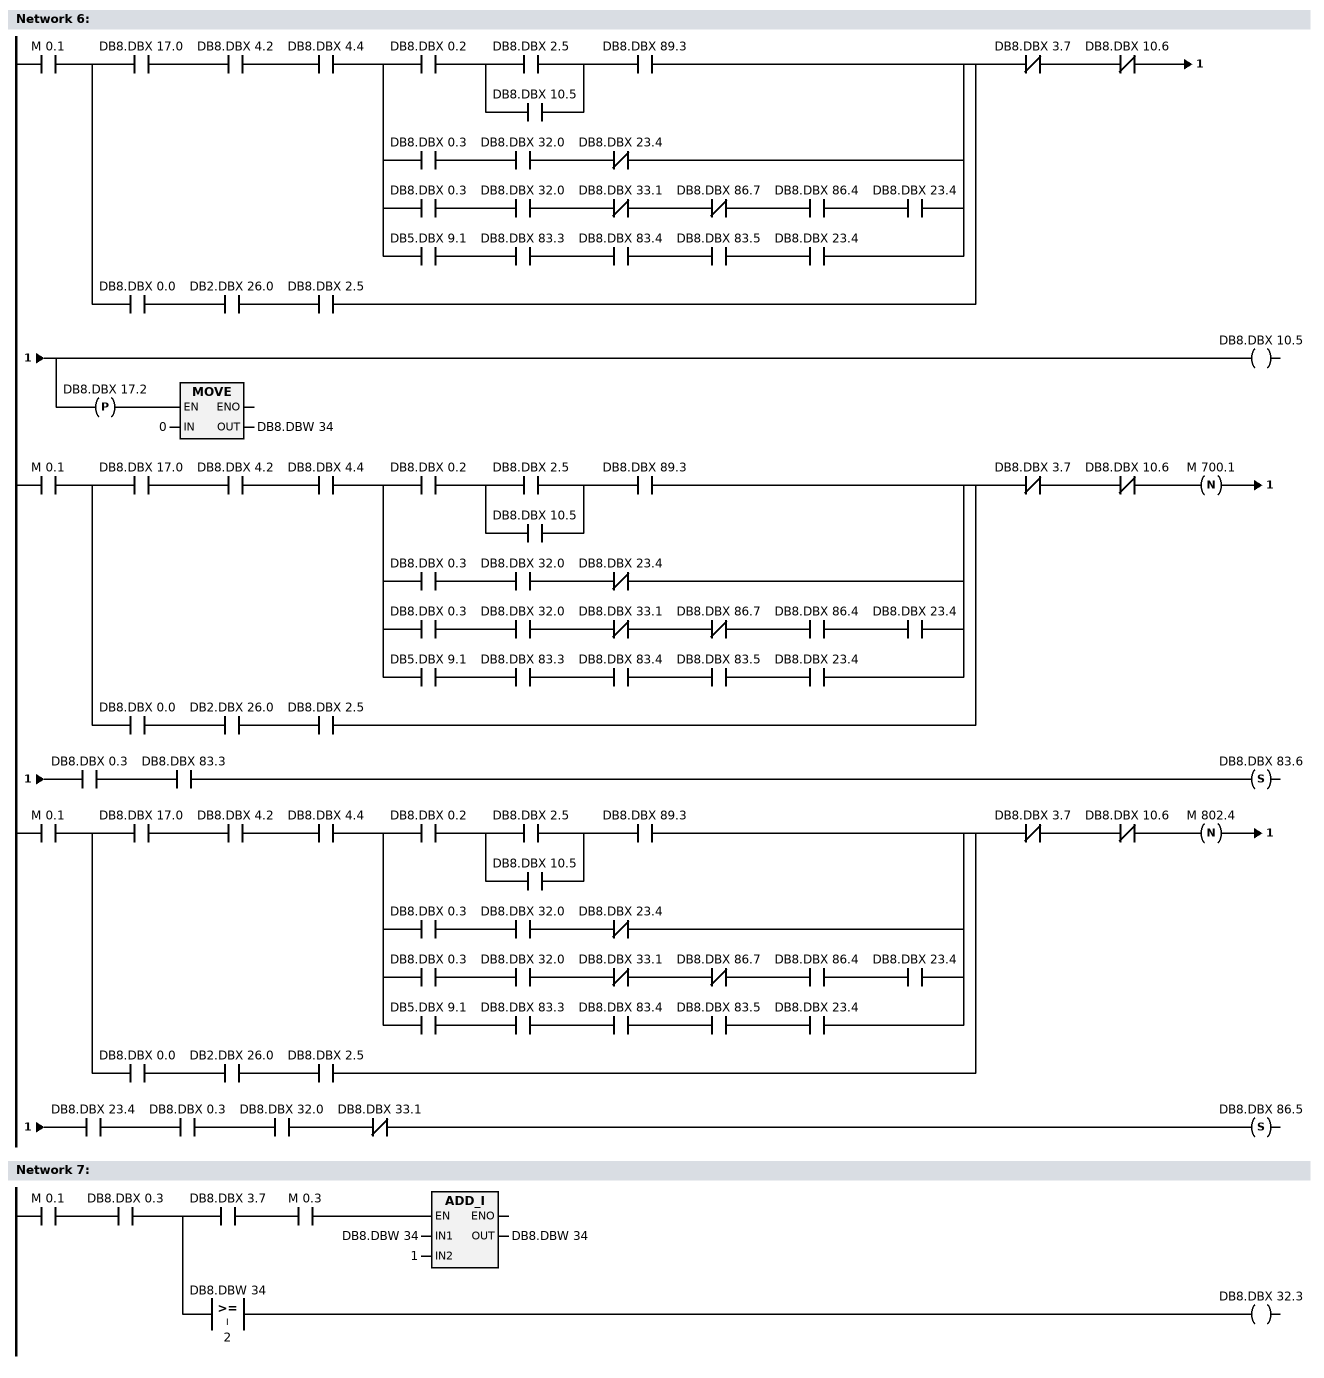
NETWORK
TITLE =
      A     M 0.1;
      A(;
      A     DB8.DBX 17.0;
      A     DB8.DBX 4.2;
      A     DB8.DBX 4.4;
      A(;
      A     DB8.DBX 0.2;
      A(;
      O     DB8.DBX 2.5;
      O     DB8.DBX 10.5;
      );
      A     DB8.DBX 89.3;
      O;
      A     DB8.DBX 0.3;
      A     DB8.DBX 32.0;
      AN    DB8.DBX 23.4;
      O;
      A     DB8.DBX 0.3;
      A     DB8.DBX 32.0;
      AN    DB8.DBX 33.1;
      AN    DB8.DBX 86.7;
      A     DB8.DBX 86.4;
      A     DB8.DBX 23.4;
      O;
      A     DB5.DBX 9.1;
      A     DB8.DBX 83.3;
      A     DB8.DBX 83.4;
      A     DB8.DBX 83.5;
      A     DB8.DBX 23.4;
      );
      O;
      A     DB8.DBX 0.0;
      A     DB2.DBX 26.0;
      A     DB8.DBX 2.5;
      );
      AN    DB8.DBX 3.7;
      AN    DB8.DBX 10.6;
      =     L 0.0;
      A     L 0.0;
      BLD   102;
      =     DB8.DBX 10.5;
      A     L 0.0;
      FP    DB8.DBX 17.2;
      JNB   M001;
      L     0;
      T     DB8.DBW 34;
M001: NOP   0;
      A(;
      A     L 0.0;
      FN    M 700.1;
      );
      A     DB8.DBX 0.3;
      A     DB8.DBX 83.3;
      S     DB8.DBX 83.6;
      A(;
      A     L 0.0;
      FN    M 802.4;
      );
      A     DB8.DBX 23.4;
      A     DB8.DBX 0.3;
      A     DB8.DBX 32.0;
      AN    DB8.DBX 33.1;
      S     DB8.DBX 86.5;
NETWORK
TITLE =
      A     M 0.1;
      A     DB8.DBX 0.3;
      =     L 0.0;
      A     L 0.0;
      A     DB8.DBX 3.7;
      A     M 0.3;
      JNB   M002;
      L     DB8.DBW 34;
      L     1;
      +I;
      T     DB8.DBW 34;
M002: NOP   0;
      A     L 0.0;
      A(;
      L     DB8.DBW 34;
      L     2;
      >=I;
      );
      =     DB8.DBX 32.3;
